# B&R Automation Studio project EFI (part 23)

#### SafetySample.var
```iecst
(********************************************************************
 * COPYRIGHT -- Bernecker + Rainer
 ********************************************************************
 * Program: SafetySample
 * File: SafetySample.var
 * Author: B&R
 ********************************************************************
 * Local variables of program SafetySample
 ********************************************************************)
VAR
	appcmd1 : DownloadCmdApplicationTypeV1; (*command structure for application download*)
	dataAcknMachineOptions : DownloadAcknMaOpTypeV1; (*data to acknowledge bit machine options*)
	datacmd1 : DownloadCmdMaOpTypeV1; (*command structure for machine options download*)
	datacmd2 : DownloadCmdExtMaOpTypeV1; (*command structure for extended machine options download*)
	dataMachineOptionsBitInput : ConfigurationBitOptionsTypeV1; (*data for bit machine options*)
	dataModuleFlagsInput : ConfigurationModuleFlagsTypeV1; (*data for module flags*)
	dialogApplication : BOOL; (*visualization dialog for application download*)
	dialogButtonLeft : BOOL; (*left button in visualization dialog*)
	dialogButtonRight : BOOL; (*right button in visualization dialog*)
	dialogData : BOOL; (*visualization dialog for machine options download*)
	dialogExtData : BOOL; (*visualization dialog for extended machine options download*)
	dialogRemoteCmd : BOOL; (*visualization dialog for remote control*)
	executeapp1 : BOOL; (*execute application download*)
	executedata1 : BOOL; (*execute machine options download*)
	executedata2 : BOOL; (*execute extended machine options download*)
	executeRemoteCmd : BOOL; (*execute remote control*)
	indexButtonLeft : UINT; (*index for button text*)
	indexButtonRight : UINT; (* index for button text*)
	indexCompareTextData : UINT; (*index for compare message machine options*)
	indexCompareTextExtData : UINT; (*index for compare message extended machine options*)
	indexFAILLed : UINT; (*index FAIL led*)
	indexFwAcknLed : UINT; (*index FW-ACKN led*)
	indexHeaderText : UINT; (*index dialog header text*)
	indexMessageText : UINT; (*index message text*)
	indexMxchgLed : UINT; (*index MXCHG led*)
	indexRELed : UINT; (*index R/E led*)
	Interface : STRING[80] := 'IF3'; (*interface information for SafeLOGIC*)
	Node : USINT := 10; (*node information for SafeLOGIC*)
	pDeviceListOut : REFERENCE TO ARRAY[0..1] OF ConfigurationDeviceTypeV1; (*device list from FUB*)
	pMachineOptionsBitOut : REFERENCE TO ConfigurationBitOptionsTypeV1; (*bit machine options from FUB*)
	pModuleFlagsOut : REFERENCE TO ConfigurationModuleFlagsTypeV1; (*module flags form FUB*)
	readUDIDhighSL : EplSDORead; (*function block to read UDID high from device*)
	readUDIDhighSLX : AsIOAccRead; (*function block to read UDID high from device*)
	readUDIDlowSL : EplSDORead; (*function block to read UDID low from device*)
	readUDIDlowSLX : AsIOAccRead; (*function block to read UDID low from device*)
	remotecmd : RemoteControlCmdTypeV1; (*command structure for remote control*)
	safeDownloadApplication_0 : safeDownloadApplication; (*function block safeDownloadApplication*)
	safeDownloadData_0 : safeDownloadData; (*function block safeDownloadData*)
	safeDownloadData_1 : safeDownloadData; (*function block safeDownloadData*)
	safeRemoteControl_0 : safeRemoteControl; (*function block safeRemoteControl*)
	slxused : BOOL; (*SafeLOGIC-X is used*)
	Station : STRING[80] := 'IF6.ST3'; (*station information for SafeLOGIC-X*)
	statusAcknInfoData : UINT; (*acknowledge boxes for machine options*)
	statusAcknInfoExtData : UINT; (*acknowledge boxes for extended machine options*)
	statusButtonActiv : ARRAY[0..15] OF USINT; (*button activ*)
	statusButtonInactiv : ARRAY[0..15] OF USINT; (*button inactiv*)
	statusButtonUnlockApp : UINT; (*unlock buttons application*)
	statusButtonUnlockData : UINT; (*unlock buttons data*)
	statusButtonUnlockExtData : UINT; (*unlock buttons extended data*)
	statusDialog : UINT; (*dialog box*)
	statusSetPassword : UINT; (*visualization status to set password*)
	statusSLInformation : UINT; (*display information for SafeLOGIC*)
	stautsSLXInformation : UINT; (*display information for SafeLOGIC-X*)
	UDID_High : UINT; (*UDID_high for SafelOGIC*)
	UDID_Low : UDINT; (*UDID_low for SafeLOGIC*)
	visuAcknExtData : DownloadAcknExtMaOpTypeV1; (*acknowledge extended machine options*)
	visuAcknMachineOptions : ARRAY[0..511] OF BOOL; (*acknowledge machine options*)
	visuApplicationCRC : STRING[8]; (*CRC HEX string for visualization*)
	visuDeviceListInput : ARRAY[0..1] OF DownloadDeviceTypeV1; (*device list input*)
	visuDeviceListOutput : ARRAY[0..1] OF DownloadDeviceTypeV1; (*device list output*)
	visuDintInput : ConfigurationDintOptionsTypeV1; (*DINT channels input*)
	visuDintOutput : ConfigurationDintOptionsTypeV1; (*DINT channels output*)
	visuEnableDINTOptions : BOOL; (*enable DINT options*)
	visuEnableINTOptions : BOOL; (*enable INT options*)
	visuEnableMachineOptions : BOOL; (*enable BIT options*)
	visuEnableModuleFlags : BOOL; (*enable module flags*)
	visuEnableUDINTOptions : BOOL; (*enable UDINT options*)
	visuEnableUINTOptions : BOOL; (*enable UINT options*)
	visuIntInput : ConfigurationIntOptionsTypeV1; (*INT channels input*)
	visuIntOutput : ConfigurationIntOptionsTypeV1; (*INT channels output*)
	visuMachineOptionsBitInput : ARRAY[0..511] OF BOOL; (*BIT options input*)
	visuMachineOptionsBitOutput : ARRAY[0..511] OF BOOL; (*BIT options output*)
	visuModuleFlagsNotPresentInput : ARRAY[0..1023] OF BOOL; (*not present module flags input*)
	visuModuleFlagsNotPresentOutput : ARRAY[0..1023] OF BOOL; (*not present module flags output*)
	visuModuleFlagsOptionalInput : ARRAY[0..1023] OF BOOL; (*optional module flags input*)
	visuModuleFlagsOptionalOutput : ARRAY[0..1023] OF BOOL; (*optional module flags output*)
	visuModuleFlagsStartupInput : ARRAY[0..1023] OF BOOL; (*startup module flags input*)
	visuModuleFlagsStartupOutput : ARRAY[0..1023] OF BOOL; (*startup module flags output*)
	visuUDID_High : STRING[8]; (*UDID hex string for visualization*)
	visuUDID_Low : STRING[8]; (*UDID hex string for visualization*)
	visuUdintInput : ConfigurationUdintOptionsTypeV1; (*UDINT channels input*)
	visuUdintOutput : ConfigurationUdintOptionsTypeV1; (*UDINT channels output*)
	visuUintInput : ConfigurationUintOptionsTypeV1; (*UINT channels input*)
	visuUintOutput : ConfigurationUintOptionsTypeV1; (*UINT channels output*)
	visuUsedSLIDData : UINT; (*SafeLOGIC ID for data download*)
	visuUsedSLIDRemote : UINT; (*SafeLOGIC ID for remote control*)
	xcnt : UINT; (*counter variable*)
	xEnableSafetyProgram : BOOL := FALSE; (*By default, it is not running*)
END_VAR
```

#### SafetySample.fun
```iecst
(********************************************************************
 * COPYRIGHT -- Bernecker + Rainer
 ********************************************************************
 * Program: SafetySample
 * File: SafetySample.fun
 * Author: B&R
 ********************************************************************
 * Functions and function blocks of program SafetySample
 ********************************************************************)

FUNCTION itoahex : UINT (*converts a UDINT values into a HEX character string*) (*$GROUP=User*)
	VAR_INPUT
		value : UDINT; (*UDINT value to be converted into a HEX character string*)
		pString : UDINT; (*pointer to the destination character string*)
	END_VAR
	VAR
		i_counter : USINT; (*internal variable*)
		i_value : UDINT; (*internal variable*)
		i_cvalue : USINT; (*internal variable*)
	END_VAR
END_FUNCTION
```

#### itoahex.st
```iecst
(********************************************************************
 * COPYRIGHT -- Bernecker + Rainer
 ********************************************************************
 * Program: SafetySample
 * File: itoahex.st
 * Author: B&R
 ********************************************************************
 * Implementation of program SafetySample
 ********************************************************************)

(* converts a UDINT values into a HEX character string *)
FUNCTION itoahex

	i_value := value;

	FOR i_counter := 0 TO 7 BY 1  DO
		i_cvalue := REAL_TO_USINT(brmfloor(UDINT_TO_REAL(i_value / REAL_TO_UDINT(EXPT(16, 7 - i_counter)))));
		IF i_cvalue = 0 THEN
			brsmemset(pString + i_counter, 48, 1); // 48 Dec = ASCII '0'
		ELSIF i_cvalue > 0 AND i_cvalue < 10 THEN
			brsitoa(i_cvalue, pString + i_counter);
		ELSIF i_cvalue >= 10 THEN
			brsmemset(pString + i_counter, i_cvalue + 55, 1); // 65 Dec = ASCII 'A'
		END_IF

		IF i_cvalue > 0 THEN
			i_value := i_value - REAL_TO_UDINT(EXPT(16, 7 - i_counter)) * i_cvalue;
		END_IF

	END_FOR

	itoahex := 0;

END_FUNCTION
```

#### SafetySample.st
```iecst
(********************************************************************
 * COPYRIGHT -- Bernecker + Rainer
 ********************************************************************
 * Program: SafetySample
 * File: SafetySample.st
 * Author: B&R
 ********************************************************************
 * Implementation of program SafetySample
 ********************************************************************)

PROGRAM _INIT

(* command structure for remote control FUB *)
remotecmd.Version := safeVERSION_R107;	(* version *)
remotecmd.Password := '';				(* password *)

(* command structure for application download *)
appcmd1.Version := safeVERSION_R107;	(* version *)
appcmd1.Password := '';					(* password *)
appcmd1.ApplicationID := 1;				(* application id *)

(* command structure for machine options download *)
datacmd1.Version := safeVERSION_R107;								(* version *)
datacmd1.Password := '';											(* password *)
datacmd1.pDeviceListInput := ADR(visuDeviceListInput);				(* device list *)
datacmd1.pMachineOptionsInput := ADR(dataMachineOptionsBitInput);	(* bit machine options *)
datacmd1.pModuleFlagsInput := ADR(dataModuleFlagsInput);			(* module flags *)
datacmd1.pAcknMachineOptions := ADR(dataAcknMachineOptions);		(* acknowledge information *)

(* command structure for extended machine options *)
datacmd2.Version := safeVERSION_R107;					(* version *)
datacmd2.Password := '';								(* password *)
datacmd2.pIntDataInput := ADR(visuIntInput);			(* INT channels *)
datacmd2.NumberIntInput := 1;							(* number of INT channels *)
datacmd2.pUintDataInput := ADR(visuUintInput);			(* UINT channels *)
datacmd2.NumberUintInput := 1;							(* number of UINT channels *)
datacmd2.pDintDataInput := ADR(visuDintInput);			(* DINT channels *)
datacmd2.NumberDintInput := 1;							(* number of DINT channels *)
datacmd2.pUdintDataInput := ADR(visuUdintInput);		(* UDINT channels *)
datacmd2.NumberUdintInput := 1;							(* number of UDINT channels *)
datacmd2.pAcknMachineOptions := ADR(visuAcknExtData);	(* acknowledge information *)

(* hide elements in visualization *)
FOR xcnt := 0 TO SIZEOF(statusButtonActiv) - 1 DO
	statusButtonActiv[xcnt] := 1;
END_FOR

(* hide elements in visualization *)
statusButtonUnlockApp := 1;
statusButtonUnlockData := 1;
statusAcknInfoData := 1;
statusButtonUnlockExtData := 1;
statusAcknInfoExtData := 1;
statusDialog := 1;

(* set SafeLOGIC ID *)
visuUsedSLIDRemote := 1;
visuUsedSLIDData := 1;

END_PROGRAM

PROGRAM _CYCLIC

	IF NOT xEnableSafetyProgram THEN
		RETURN;
	END_IF

	(****************************************************************************************************************************************)
	(****************************************************************************************************************************************)
	(****************************************************************************************************************************************)
	(* show dialog to ackn command *)
	IF (dialogRemoteCmd = 1) THEN
		statusDialog := 0;
		dialogRemoteCmd := 0;
		indexButtonLeft := 0;
		indexButtonRight := 1;
		indexHeaderText := 0;
		IF (remotecmd.Data = safeCMD_SK_FORMAT) THEN
			indexMessageText := 0;
		ELSIF (remotecmd.Data = safeCMD_SK_XCHG) THEN
			indexMessageText := 1;
		ELSIF (remotecmd.Data = safeCMD_1_UDID_ACKN) THEN
			indexMessageText := 2;
		ELSIF (remotecmd.Data = safeCMD_2_UDID_ACKN) THEN
			indexMessageText := 3;
		ELSIF (remotecmd.Data = safeCMD_3_UDID_ACKN) THEN
			indexMessageText := 4;
		ELSIF (remotecmd.Data = safeCMD_4_UDID_ACKN) THEN
			indexMessageText := 5;
		ELSIF (remotecmd.Data =  safeCMD_N_UDID_ACKN) THEN
			indexMessageText := 6;
		ELSIF (remotecmd.Data =  safeCMD_CLEAR_DATA) THEN
			indexMessageText := 7;
		ELSIF (remotecmd.Data = safeCMD_FW_ACKN) THEN
			indexMessageText := 8;
		ELSIF (remotecmd.Data = safeCMD_RESET) THEN
			indexMessageText := 9;
		END_IF
	END_IF

	(* if dialog is ackn execute fub *)
	IF (dialogButtonLeft = 1 AND indexHeaderText = 0) THEN
		executeRemoteCmd := 1;
		dialogButtonLeft := 0;
		statusDialog := 1;
	ELSIF (dialogButtonRight = 1 AND indexHeaderText = 0) THEN
		dialogButtonRight := 0;
		statusDialog := 1;
	END_IF

	(* password must be at least 6 characters long *)
	IF brsstrlen(ADR(remotecmd.NewPassword)) < 6 THEN
		statusSetPassword := 2;
	ELSE
		statusSetPassword := 0;
	END_IF

	safeRemoteControl_0(SafeLOGICID := visuUsedSLIDRemote, Execute := executeRemoteCmd, pCommandData := ADR(remotecmd));
	(* reset execution flag *)
	IF (safeRemoteControl_0.Done = 1 OR safeRemoteControl_0.Error = 1) THEN
		executeRemoteCmd := 0;
	END_IF

	(* variables for visualization *)
	IF (safeRemoteControl_0.SafeLOGICStatus.SafeKEYChanged = 1) THEN
		FOR xcnt := 0 TO SIZEOF(statusButtonActiv) - 1 DO
			statusButtonActiv[xcnt] := 1;
 			statusButtonInactiv[xcnt] := 0;
		END_FOR
		statusButtonActiv[1] := 0;
 		statusButtonInactiv[1] := 1;
	ELSIF (safeRemoteControl_0.SafeLOGICStatus.NumberOfUDIDMismatches = 1 AND safeRemoteControl_0.SafeLOGICStatus.Scanning = 0) THEN
		FOR xcnt := 0 TO SIZEOF(statusButtonActiv) - 1 DO
			statusButtonActiv[xcnt] := 1;
 			statusButtonInactiv[xcnt] := 0;
		END_FOR
		statusButtonActiv[3] := 0;
 		statusButtonInactiv[3] := 1;
	ELSIF (safeRemoteControl_0.SafeLOGICStatus.NumberOfUDIDMismatches = 2 AND safeRemoteControl_0.SafeLOGICStatus.Scanning = 0) THEN
		FOR xcnt := 0 TO SIZEOF(statusButtonActiv) - 1 DO
			statusButtonActiv[xcnt] := 1;
 			statusButtonInactiv[xcnt] := 0;
		END_FOR
		statusButtonActiv[4] := 0;
 		statusButtonInactiv[4] := 1;
	ELSIF (safeRemoteControl_0.SafeLOGICStatus.NumberOfUDIDMismatches = 3 AND safeRemoteControl_0.SafeLOGICStatus.Scanning = 0) THEN
		FOR xcnt := 0 TO SIZEOF(statusButtonActiv) - 1 DO
			statusButtonActiv[xcnt] := 1;
 			statusButtonInactiv[xcnt] := 0;
		END_FOR
		statusButtonActiv[5] := 0;
 		statusButtonInactiv[5] := 1;
	ELSIF (safeRemoteControl_0.SafeLOGICStatus.NumberOfUDIDMismatches = 4 AND safeRemoteControl_0.SafeLOGICStatus.Scanning = 0) THEN
		FOR xcnt := 0 TO SIZEOF(statusButtonActiv) - 1 DO
			statusButtonActiv[xcnt] := 1;
 			statusButtonInactiv[xcnt] := 0;
		END_FOR
		statusButtonActiv[6] := 0;
 		statusButtonInactiv[6] := 1;
	ELSIF (safeRemoteControl_0.SafeLOGICStatus.NumberOfUDIDMismatches > 4 AND safeRemoteControl_0.SafeLOGICStatus.Scanning = 0) THEN
		FOR xcnt := 0 TO SIZEOF(statusButtonActiv) - 1 DO
			statusButtonActiv[xcnt] := 1;
 			statusButtonInactiv[xcnt] := 0;
		END_FOR
		statusButtonActiv[7] := 0;
 		statusButtonInactiv[7] := 1;
	ELSIF (safeRemoteControl_0.SafeLOGICStatus.NumberOfDifferentFirmware <> 0 AND safeRemoteControl_0.SafeLOGICStatus.Scanning = 0) THEN
		FOR xcnt := 0 TO SIZEOF(statusButtonActiv) - 1 DO
			statusButtonActiv[xcnt] := 1;
 			statusButtonInactiv[xcnt] := 0;
		END_FOR
		statusButtonActiv[11] := 0;
 		statusButtonInactiv[11] := 1;
	ELSE
		FOR xcnt := 0 TO SIZEOF(statusButtonActiv) - 1 DO
			statusButtonActiv[xcnt] := 1;
 			statusButtonInactiv[xcnt] := 0;
		END_FOR
	END_IF
	(* status text - MXCHG *)
	IF (safeRemoteControl_0.SafeLOGICStatus.LedTestActive = 1) THEN
		indexMxchgLed := 40;
	ELSIF (safeRemoteControl_0.SafeLOGICStatus.Scanning = 1) THEN
		indexMxchgLed := 30;
	ELSIF (safeRemoteControl_0.SafeLOGICStatus.NumberOfUDIDMismatches = 1) THEN
		indexMxchgLed := 1;
	ELSIF (safeRemoteControl_0.SafeLOGICStatus.NumberOfUDIDMismatches = 2) THEN
		indexMxchgLed := 2;
	ELSIF (safeRemoteControl_0.SafeLOGICStatus.NumberOfUDIDMismatches = 3) THEN
		indexMxchgLed := 3;
	ELSIF (safeRemoteControl_0.SafeLOGICStatus.NumberOfUDIDMismatches = 4) THEN
		indexMxchgLed := 4;
	ELSIF (safeRemoteControl_0.SafeLOGICStatus.NumberOfUDIDMismatches > 4) THEN
		indexMxchgLed := 5;
	ELSIF (safeRemoteControl_0.SafeLOGICStatus.NumberOfMissingModules <> 0) THEN
		indexMxchgLed := 20;
	ELSIF (safeRemoteControl_0.SafeLOGICStatus.NumberOfUDIDMismatches = 0) THEN
		indexMxchgLed := 10;
	END_IF
	(* status text - FW-ACKN *)
	IF (safeRemoteControl_0.SafeLOGICStatus.SafeKEYChanged = 0 AND safeRemoteControl_0.SafeLOGICStatus.NumberOfDifferentFirmware = 0) THEN
		indexFwAcknLed := 10;
	ELSIF (safeRemoteControl_0.SafeLOGICStatus.SafeKEYChanged = 1) THEN
		indexFwAcknLed := 1;
	ELSIF (safeRemoteControl_0.SafeLOGICStatus.NumberOfDifferentFirmware <> 0) THEN
		indexFwAcknLed := 2;
	END_IF
	(* status text - FAIL *)
	IF (safeRemoteControl_0.SafeLOGICStatus.FailSafe <> 16#55) THEN
		indexFAILLed := 2;
	ELSIF (safeRemoteControl_0.SafeLOGICStatus.openSAFETYstate = 0) THEN
		indexFAILLed := 0;
	ELSIF (safeRemoteControl_0.SafeLOGICStatus.openSAFETYstate = 1) THEN
		indexFAILLed := 1;
	END_IF
	(* status text - R/E *)
	indexRELed := safeRemoteControl_0.SafeLOGICStatus.SafeOSState;

	(****************************************************************************************************************************************)
	(****************************************************************************************************************************************)
	(****************************************************************************************************************************************)
	(* show dialog to ackn command *)
	IF (dialogApplication = 1) THEN
		statusDialog := 0;
		dialogApplication := 0;
		indexButtonLeft := 0;
		indexButtonRight := 1;
		indexHeaderText := 1;
		indexMessageText := 10;
	END_IF

	(* if dialog is ackn unlock application *)
	IF (dialogButtonLeft = 1 AND indexHeaderText = 1) THEN
		appcmd1.Unlock := 1;
		dialogButtonLeft := 0;
		statusDialog := 1;
	ELSIF (dialogButtonRight = 1 AND indexHeaderText = 1) THEN
		appcmd1.Unlock := 2;
		dialogButtonRight := 0;
		statusDialog := 1;
	END_IF

	(* convert application CRC to HEX string *)
	itoahex(safeDownloadApplication_0.ApplicationCRC, ADR(visuApplicationCRC));

	safeDownloadApplication_0(SafeLOGICID := appcmd1.ApplicationID, Execute := executeapp1, pCommandData := ADR(appcmd1));

	(* show unlock button *)
	IF (safeDownloadApplication_0.UnlockRequired = 1) THEN
		statusButtonUnlockApp := 0;
	ELSE
		appcmd1.Unlock := 0;
		statusButtonUnlockApp := 1;
	END_IF

	(****************************************************************************************************************************************)
	(****************************************************************************************************************************************)
	(****************************************************************************************************************************************)
	(* disable machine options *)
	IF (visuEnableMachineOptions = FALSE) THEN
		datacmd1.pMachineOptionsInput := 0;
	ELSE
		datacmd1.pMachineOptionsInput := ADR(dataMachineOptionsBitInput);
	END_IF

	(* disable module flags *)
	IF (visuEnableModuleFlags = FALSE) THEN
		datacmd1.pModuleFlagsInput := 0;
	ELSE
		datacmd1.pModuleFlagsInput := ADR(dataModuleFlagsInput);
	END_IF

	(* Machine Option Bit #000 *)
	IF (visuMachineOptionsBitInput[0] = 1) THEN
		dataMachineOptionsBitInput.BitData[0].0 := 1;
	ELSE
		dataMachineOptionsBitInput.BitData[0].0 := 0;
	END_IF
	(* Machine Option Bit #001 *)
	IF (visuMachineOptionsBitInput[1] = 1) THEN
		dataMachineOptionsBitInput.BitData[0].1 := 1;
	ELSE
		dataMachineOptionsBitInput.BitData[0].1 := 0;
	END_IF
	(* Machine Option Bit #002 *)
	IF (visuMachineOptionsBitInput[2] = 1) THEN
		dataMachineOptionsBitInput.BitData[0].2 := 1;
	ELSE
		dataMachineOptionsBitInput.BitData[0].2 := 0;
	END_IF
	(* Optional Flag Module #1 *)
	IF (visuModuleFlagsOptionalInput[1] = 1) THEN
		dataModuleFlagsInput.Optional[0].1 := 1;
	ELSE
		dataModuleFlagsInput.Optional[0].1 := 0;
	END_IF
	(* Optional Flag Module #2 *)
	IF (visuModuleFlagsOptionalInput[2] = 1) THEN
		dataModuleFlagsInput.Optional[0].2 := 1;
	ELSE
		dataModuleFlagsInput.Optional[0].2 := 0;
	END_IF
	(* Startup Flag Module #1 *)
	IF (visuModuleFlagsStartupInput[1] = 1) THEN
		dataModuleFlagsInput.Startup[0].1 := 1;
	ELSE
		dataModuleFlagsInput.Startup[0].1 := 0;
	END_IF
	(* Startup Flag Module #2 *)
	IF (visuModuleFlagsStartupInput[2] = 1) THEN
		dataModuleFlagsInput.Startup[0].2 := 1;
	ELSE
		dataModuleFlagsInput.Startup[0].2 := 0;
	END_IF
	(* Not_Present Flag Module #1 *)
	IF (visuModuleFlagsNotPresentInput[1] = 1) THEN
		dataModuleFlagsInput.NotPresent[0].1 := 1;
	ELSE
		dataModuleFlagsInput.NotPresent[0].1 := 0;
	END_IF
	(* Not_Present Flag Module #2 *)
	IF (visuModuleFlagsNotPresentInput[2] = 1) THEN
		dataModuleFlagsInput.NotPresent[0].2 := 1;
	ELSE
		dataModuleFlagsInput.NotPresent[0].2 := 0;
	END_IF

	(* Ackn Machine Option Bit #000 *)
	IF (visuAcknMachineOptions[0] = 1) THEN
		dataAcknMachineOptions.AcknBitOptions[0].0 := 1;
	ELSE
		dataAcknMachineOptions.AcknBitOptions[0].0 := 0;
	END_IF
	(* Ackn Machine Option Bit #001 *)
	IF (visuAcknMachineOptions[1] = 1) THEN
		dataAcknMachineOptions.AcknBitOptions[0].1 := 1;
	ELSE
		dataAcknMachineOptions.AcknBitOptions[0].1 := 0;
	END_IF
	(* Ackn Machine Option Bit #002 *)
	IF (visuAcknMachineOptions[2] = 1) THEN
		dataAcknMachineOptions.AcknBitOptions[0].2 := 1;
	ELSE
		dataAcknMachineOptions.AcknBitOptions[0].2 := 0;
	END_IF

	(* show dialog to ackn command *)
	IF (dialogData = 1) THEN
		statusDialog := 0;
		dialogData := 0;
		indexButtonLeft := 0;
		indexButtonRight := 1;
		indexHeaderText := 2;
		indexMessageText := 11;
	END_IF

	(* if dialog is ackn unlock data *)
	IF (dialogButtonLeft = 1 AND indexHeaderText = 2) THEN
		datacmd1.Unlock := 1;
		dialogButtonLeft := 0;
		statusDialog := 1;
	ELSIF (dialogButtonRight = 1 AND indexHeaderText = 2) THEN
		datacmd1.Unlock := 2;
		dialogButtonRight := 0;
		statusDialog := 1;
	END_IF

	safeDownloadData_0(SafeLOGICID := visuUsedSLIDData, Execute := executedata1, Type:= safeDATA_TYPE_MAOP, pCommandData := ADR(datacmd1));

	(* data compare failed *)
	IF (safeDownloadData_0.StatusID = safeERR_DL_COMPARE_FAILED) THEN
		indexCompareTextData := 2;
	ELSE
		indexCompareTextData := 0;
	END_IF

	IF (safeDownloadData_0.UnlockRequired = 1) THEN
		(* data compare successful *)
		indexCompareTextData := 1;
		IF (datacmd1.pDeviceListOutput <> 0 AND datacmd1.NumberDevicesOutput <> 0) THEN
			pDeviceListOut ACCESS datacmd1.pDeviceListOutput;

			(* device #1 *)
			visuDeviceListOutput[0].SADR := pDeviceListOut[0].SADR;
			brsmemcpy(ADR(visuDeviceListOutput[0].UDID_High), ADR(pDeviceListOut[0].UDID[0]), 2);
			(* swap UDID *)
			visuDeviceListOutput[0].UDID_High := swapUINT(visuDeviceListOutput[0].UDID_High);
			brsmemcpy(ADR(visuDeviceListOutput[0].UDID_Low), ADR(pDeviceListOut[0].UDID[2]), 4);
			(* swap UDID *)
			visuDeviceListOutput[0].UDID_Low := swapUDINT(visuDeviceListOutput[0].UDID_Low);
			(* device #2 *)
			visuDeviceListOutput[1].SADR := pDeviceListOut[1].SADR;
			brsmemcpy(ADR(visuDeviceListOutput[1].UDID_High), ADR(pDeviceListOut[1].UDID[0]), 2);
			(* swap UDID *)
			visuDeviceListOutput[1].UDID_High := swapUINT(visuDeviceListOutput[1].UDID_High);
			brsmemcpy(ADR(visuDeviceListOutput[1].UDID_Low), ADR(pDeviceListOut[1].UDID[2]), 4);
			(* swap UDID *)
			visuDeviceListOutput[1].UDID_Low := swapUDINT(visuDeviceListOutput[1].UDID_Low);
		END_IF

		IF (datacmd1.pMachineOptionsOutput <> 0) THEN
			pMachineOptionsBitOut ACCESS datacmd1.pMachineOptionsOutput;

			(* Machine Option Bit #000 *)
			IF (pMachineOptionsBitOut.BitData[0].0 = 1) THEN
				visuMachineOptionsBitOutput[0] := 1;
			END_IF
			(* Machine Option Bit #001 *)
			IF (pMachineOptionsBitOut.BitData[0].1 = 1) THEN
				visuMachineOptionsBitOutput[1] := 1;
			END_IF
			(* Machine Option Bit #002 *)
			IF (pMachineOptionsBitOut.BitData[0].2 = 1) THEN
				visuMachineOptionsBitOutput[2] := 1;
			END_IF
		END_IF

		IF (datacmd1.pModuleFlagsOutput <> 0) THEN
			pModuleFlagsOut ACCESS datacmd1.pModuleFlagsOutput;

			(* Optional Flag Module #1 *)
			IF (pModuleFlagsOut.Optional[0].1 = 1) THEN
				visuModuleFlagsOptionalOutput[1] := 1;
			END_IF
			(* Optional Flag Module #2 *)
			IF (pModuleFlagsOut.Optional[0].2 = 1) THEN
				visuModuleFlagsOptionalOutput[2] := 1;
			END_IF
			(* Startup Flag Module #1 *)
			IF (pModuleFlagsOut.Startup[0].1 = 1) THEN
				visuModuleFlagsStartupOutput[1] := 1;
			END_IF
			(* Startup Flag Module #2 *)
			IF (pModuleFlagsOut.Startup[0].2 = 1) THEN
				visuModuleFlagsStartupOutput[2] := 1;
			END_IF
			(* Not_Present Flag Module #1 *)
			IF (pModuleFlagsOut.NotPresent[0].1 = 1) THEN
				visuModuleFlagsNotPresentOutput[1] := 1;
			END_IF
			(* Not_Present Flag Module #2 *)
			IF (pModuleFlagsOut.NotPresent[0].2 = 1) THEN
				visuModuleFlagsNotPresentOutput[2] := 1;
			END_IF
		END_IF
		(* show ackn box *)
		statusAcknInfoData := 0;
		(* show unlock button unlocked if one ACK is set *)
		IF (visuAcknMachineOptions[0] = 1 OR visuAcknMachineOptions[1] = 1 OR visuAcknMachineOptions[2] = 1) THEN
			statusButtonUnlockData := 0;
		END_IF
	ELSIF (safeDownloadData_0.Done = 1 OR safeDownloadData_0.Error = 1) THEN
		(* reset visualization elements *)
		brsmemset(ADR(visuDeviceListOutput), 0, SIZEOF(visuDeviceListOutput));
		brsmemset(ADR(visuMachineOptionsBitOutput), 0, SIZEOF(visuMachineOptionsBitOutput));
		brsmemset(ADR(visuModuleFlagsOptionalOutput), 0, SIZEOF(visuModuleFlagsOptionalOutput));
		brsmemset(ADR(visuModuleFlagsStartupOutput), 0, SIZEOF(visuModuleFlagsStartupOutput));
		brsmemset(ADR(visuModuleFlagsNotPresentOutput), 0, SIZEOF(visuModuleFlagsNotPresentOutput));
		(* hide ackn box *)
		statusAcknInfoData := 1;
		(* hide unlock button *)
		datacmd1.Unlock := 0;
		statusButtonUnlockData := 1;
		(* reset ackn flags *)
		visuAcknMachineOptions[0] := 0;
		visuAcknMachineOptions[1] := 0;
		visuAcknMachineOptions[2] := 0;
	ELSE
		(* hide ackn box *)
		statusAcknInfoData := 1;
		(* hide unlock button *)
		datacmd1.Unlock := 0;
		statusButtonUnlockData := 1;
	END_IF

	(****************************************************************************************************************************************)
	(****************************************************************************************************************************************)
	(****************************************************************************************************************************************)
	(* Enable for INT set *)
	IF (visuEnableINTOptions <> 0) THEN
		datacmd2.pIntDataInput := ADR(visuIntInput);
		datacmd2.NumberIntInput := 1;
	ELSE
		datacmd2.pIntDataInput := 0;
		datacmd2.NumberIntInput := 0;
	END_IF
	(* Enable for UINT set *)
	IF (visuEnableUINTOptions <> 0) THEN
		datacmd2.pUintDataInput := ADR(visuUintInput);
		datacmd2.NumberUintInput := 1;
	ELSE
		datacmd2.pUintDataInput := 0;
		datacmd2.NumberUintInput := 0;
	END_IF
	(* Enable for DINT set *)
	IF (visuEnableDINTOptions <> 0) THEN
		datacmd2.pDintDataInput := ADR(visuDintInput);
		datacmd2.NumberDintInput := 1;
	ELSE
		datacmd2.pDintDataInput := 0;
		datacmd2.NumberDintInput := 0;
	END_IF
	(* Enable for UDINT set *)
	IF (visuEnableUDINTOptions <> 0) THEN
		datacmd2.pUdintDataInput := ADR(visuUdintInput);
		datacmd2.NumberUdintInput := 1;
	ELSE
		datacmd2.pUdintDataInput := 0;
		datacmd2.NumberUdintInput := 0;
	END_IF

	(* show dialog to ackn command *)
	IF (dialogExtData = 1) THEN
		statusDialog := 0;
		dialogExtData := 0;
		indexButtonLeft := 0;
		indexButtonRight := 1;
		indexHeaderText := 3;
		indexMessageText := 11;
	END_IF

	(* if dialog is ackn unlock data *)
	IF (dialogButtonLeft = 1 AND indexHeaderText = 3) THEN
		datacmd2.Unlock := 1;
		dialogButtonLeft := 0;
		statusDialog := 1;
	ELSIF (dialogButtonRight = 1 AND indexHeaderText = 3) THEN
		datacmd2.Unlock := 2;
		dialogButtonRight := 0;
		statusDialog := 1;
	END_IF

	safeDownloadData_1(SafeLOGICID := visuUsedSLIDData, Execute := executedata2, Type:= safeDATA_TYPE_EXTMAOP, pCommandData := ADR(datacmd2));

	(* data compare failed *)
	IF (safeDownloadData_1.StatusID = safeERR_DL_COMPARE_FAILED) THEN
		indexCompareTextExtData := 2;
	ELSE
		indexCompareTextExtData := 0;
	END_IF

	IF (safeDownloadData_1.UnlockRequired = 1) THEN
		(* data compare successful *)
		indexCompareTextExtData := 1;

		(* INT channels *)
		IF (datacmd2.pIntDataOutput <> 0 AND datacmd2.NumberIntOutput <> 0) THEN
			brsmemcpy(ADR(visuIntOutput), datacmd2.pIntDataOutput, SIZEOF(visuIntOutput));
		END_IF
		(* UINT channels *)
		IF (datacmd2.pUintDataOutput <> 0 AND datacmd2.NumberUintOutput <> 0) THEN
			brsmemcpy(ADR(visuUintOutput), datacmd2.pUintDataOutput, SIZEOF(visuUintOutput));
		END_IF
		(* DINT channels *)
		IF (datacmd2.pDintDataOutput <> 0 AND datacmd2.NumberDintOutput <> 0) THEN
			brsmemcpy(ADR(visuDintOutput), datacmd2.pDintDataOutput, SIZEOF(visuDintOutput));
		END_IF
		(* UDINT channels *)
		IF (datacmd2.pUdintDataOutput <> 0 AND datacmd2.NumberUdintOutput <> 0) THEN
			brsmemcpy(ADR(visuUdintOutput), datacmd2.pUdintDataOutput, SIZEOF(visuUdintOutput));
		END_IF
		(* show ackn box *)
		statusAcknInfoExtData := 0;
		(* show unlock button if one ACK is set *)
		IF (visuAcknExtData.AcknIntOptions[0] = 1 OR visuAcknExtData.AcknUintOptions[0] = 1 OR visuAcknExtData.AcknDintOptions[0] = 1 OR visuAcknExtData.AcknUdintOptions[0] = 1) THEN
			statusButtonUnlockExtData := 0;
		END_IF
	ELSIF (safeDownloadData_1.Done = 1 OR safeDownloadData_1.Error = 1) THEN
		(* reset visualization elements *)
		brsmemset(ADR(visuIntOutput), 0, SIZEOF(visuIntOutput));
		brsmemset(ADR(visuUintOutput), 0, SIZEOF(visuUintOutput));
		brsmemset(ADR(visuDintOutput), 0, SIZEOF(visuDintOutput));
		brsmemset(ADR(visuUdintOutput), 0, SIZEOF(visuUdintOutput));
		(* hide ackn box *)
		statusAcknInfoExtData := 1;
		(* hide unlock button *)
		datacmd2.Unlock := 0;
		statusButtonUnlockExtData := 1;
		(* reset ackn flags *)
		visuAcknExtData.AcknIntOptions[0] := 0;
		visuAcknExtData.AcknUintOptions[0] := 0;
		visuAcknExtData.AcknDintOptions[0] := 0;
		visuAcknExtData.AcknUdintOptions[0] := 0;
	ELSE
		(* hide ackn box *)
		statusAcknInfoExtData := 1;
		(* hide unlock button *)
		datacmd2.Unlock := 0;
		statusButtonUnlockExtData := 1;
	END_IF

	(****************************************************************************************************************************************)
	(****************************************************************************************************************************************)
	(****************************************************************************************************************************************)
	(* read UDID from SafeLOGIC-X *)
	IF slxused = 1 THEN
		readUDIDlowSLX(enable := 1, pDeviceName := ADR(Station), pChannelName := ADR('UDID_low'));

		IF readUDIDlowSLX.status = 0 THEN
			UDID_Low := readUDIDlowSLX.value;
		ELSIF readUDIDlowSLX.status <> 65535 THEN
			UDID_Low := 0;
		END_IF

		readUDIDhighSLX(enable := 1, pDeviceName := ADR(Station), pChannelName := ADR('UDID_high'));

		IF readUDIDhighSLX.status = 0 THEN
			UDID_High := UDINT_TO_UINT(readUDIDhighSLX.value);
		ELSIF readUDIDhighSLX.status <> 65535 THEN
			UDID_High := 0;
		END_IF

		(* hide / show visualization elements *)
		stautsSLXInformation := 0;
		statusSLInformation := 1;
	(* read UDID form SafeLOGIC *)
	ELSE
		readUDIDlowSL(enable := 1, pDevice := ADR(Interface), node := Node, index := 16#2000, subindex := 6, pData := ADR(UDID_Low), datalen := SIZEOF(UDID_Low));

		IF readUDIDlowSL.status <> 0 AND readUDIDlowSL.status <> 65535 THEN
			UDID_Low := 0;
		END_IF

		readUDIDhighSL(enable := 1, pDevice := ADR(Interface), node := Node, index := 16#2000, subindex := 7, pData := ADR(UDID_High), datalen := SIZEOF(UDID_High));

		IF readUDIDhighSL.status <> 0 AND readUDIDhighSL.status <> 65535 THEN
			UDID_High := 0;
		END_IF

		(* hide / show visualization elements *)
		stautsSLXInformation := 1;
		statusSLInformation := 0;
	END_IF

	(* convert UDID to HEX string *)
	itoahex(UDID_Low, ADR(visuUDID_Low));
	itoahex(UDID_High, ADR(visuUDID_High));

	(****************************************************************************************************************************************)
	(****************************************************************************************************************************************)
	(****************************************************************************************************************************************)
	(* write UDID for SafeLOGIC to command structure *)
	appcmd1.UDID_Low := UDID_Low;
	appcmd1.UDID_High := UDID_High;
	datacmd1.UDID_Low := UDID_Low;
	datacmd1.UDID_High := UDID_High;
	datacmd2.UDID_Low := UDID_Low;
	datacmd2.UDID_High := UDID_High;

END_PROGRAM
```

- .gitignore (not shown)

### QA Notes.txt
```
This is the last folder for QA in the PLC project.
Below this folder, the QATestPLC repository have to be cloned to work properly
```

### Program Logical/UnitTest/Dryer/PrepareDryer (ANSIC) - Prepare the Machine to Start working

#### PrepareDryer.c - Groups test cases for addition
```c
/********************************************************************
 * COPYRIGHT -- Bernecker + Rainer
 ********************************************************************
 * Program: PrepareMachine
 * Author: Jorge Murria
 ********************************************************************
 * Prepare machine with basic test to allow proper behabior
 * and starting tasks
 ********************************************************************/

#include <bur/plctypes.h>

#ifdef _DEFAULT_INCLUDES
#include <AsDefault.h>
#endif

#include "UnitTest.h"

#include <stdio.h>
#include <unistd.h>
#include <time.h>         /* clock_t, clock, CLOCKS_PER_SEC */
#include <astime.h>

_LOCAL TIME TimeLast;
_LOCAL TIME endtime;
_LOCAL UDINT diff_t;
_LOCAL STRING stringAux[120];

#define FALSE 0
#define TRUE 1

void nextState(){
	exTimesPreFast = gDryer.St.exec.fast;
	exTimesPreSlow = gDryer.St.exec.slow;
	gTestsExec.iTestState++;
	TimeLast = clock_ms();
}

_TEST test_GoToZero(void)
{
	strcpy(gTestsExec.TestName, "test_GoToZero");
	switch (gTestsExec.iTestState)
	{
		case 0:
			gSimMachine.Commands.xToZero = TRUE;
			nextState();
			break;

		case 1:
			strcpy(gTestsExec.TestStateDesctiption, "Going to Zero");
			TEST_BUSY_CONDITION( !gDryer.St.Mode.xZero );
			nextState();
			break;

		case 2:
			gTestsExec.iTestState = 0;
			TEST_ASSERT(TRUE);
			TEST_DONE;
			break;

		default:
			break;
	}
}

_TEST test_PrepareBasicConfig(void)
{
	strcpy(gTestsExec.TestName, "test_PrepareBasicConfig");
	switch (gTestsExec.iTestState)
	{
		case 0:

			gDryer.Pt.SW.rBeltSpeedSetPoint = 15.0;	// 15.0m/min
			gDryer.Pt.SW.tiDelayConsent = SECONDS_TO_TIME(2);
			gDryer.In.xConsentOk = TRUE;

			gDryer.Pt.SW.Safety.rMaxBeltSpeedSetPoint = 70.0;
			gDryer.Pt.SW.Safety.rMarginSafePrint = 1.1;

			gBelt.parSw.rAxisLength = 650.0;
			gBelt.parSw.rGearBox = 35.0;

			gDryer.Pt.SW.xEnableNir = TRUE;

			gTransVacuum[1].Inputs.iPressureRaw = 16384; //This value is the equivalent to 0mbar of vacuum

			nextState();
			break;

		case 1:
			TEST_BUSY_CONDITION( gDryer.St.exec.fast < exTimesPreFast + 5 ); //We'll wait xx scan cycles
			nextState();
			break;

		case 2:
			gTestsExec.iTestState = 0;
			TEST_ASSERT(gDryer.Pt.xLeftHandMachine);
			TEST_DONE;
			break;

		default:
			break;
	}
}

_TEST test_GoToManualFromZero(void)
{
	strcpy(gTestsExec.TestName, "test_GoToManualFromZero");
	switch (gTestsExec.iTestState)
	{
		case 0:
			gSimMachine.Commands.xToZero = TRUE;
			nextState();
			break;

		case 1:
			strcpy(gTestsExec.TestStateDesctiption, "Going to Zero");
			TEST_BUSY_CONDITION( !gDryer.St.Mode.xZero );
			nextState();
			break;

		case 2:
			gSimMachine.Commands.xToManual = TRUE;
			nextState();
			break;

		case 3:
			strcpy(gTestsExec.TestStateDesctiption, "Going to Manual");
			TEST_BUSY_CONDITION( !gDryer.St.Mode.xManual );
			nextState();
			break;

		case 4:
			strcpy(gTestsExec.TestName, "test_PrepareMachine Finished!! Congrats!");
			strcpy(gTestsExec.TestStateDesctiption, "--");

			gTestsExec.iTestState = 0;
			TEST_ASSERT(TRUE);

			TEST_DONE;
			break;

		default:
			break;
	}
}

_TEST test_ReferenceManualMotors(void)
{
	if (gDryer.Pt.MachineModel != DryerType_NOZ2_NIR_ARCLAMP){
		iTestState = 0;
		TEST_DONE;
	}
	strcpy(gTestsExec.TestName, "test_ReferenceManualMotors");
	switch (gTestsExec.iTestState)
	{
		case 0:
			gSimMachine.Commands.xToManual = TRUE;
			nextState();
			break;

		case 1:
			strcpy(gTestsExec.TestStateDesctiption, "Going to Manual");
			TEST_BUSY_CONDITION( !gDryer.St.Mode.xManual );
			nextState();
			break;

		case 2:
			TEST_BUSY_CONDITION( gDryer.St.exec.fast < exTimesPreFast + 3 ); //We'll wait xx scan cycles
			gSimpleBlock[1].commands.xBarHomeOrder = TRUE;
			nextState();
			break;

		case 3:
			strcpy(gTestsExec.TestStateDesctiption, "Referencing vertical motors");
			TEST_BUSY_CONDITION( !gSimpleBlock[1].Status.Motor.xBarsHomed );
			nextState();
			break;

		case 4:
			gTestsExec.iTestState = 0;
			TEST_ASSERT(TRUE);

			strcpy(gTestsExec.TestName, "test_PrepareMachine Finished!! Congrats!");
			strcpy(gTestsExec.TestStateDesctiption, "--");

			TEST_DONE;
			break;

		default:
			break;
	}
}

/*
B+R UnitTest: This is generated code.
Do not edit! Do not move!
Description: UnitTest Testprogramm infrastructure (TestSet).
LastUpdated: 2021-05-20 08:42:32Z
By B+R UnitTest Helper Version: 2.0.1.59
*/
UNITTEST_FIXTURES(fixtures)
{
	new_TestFixture("test_GoToZero", test_GoToZero),
	new_TestFixture("test_PrepareBasicConfig", test_PrepareBasicConfig),
	new_TestFixture("test_GoToManualFromZero", test_GoToManualFromZero),
	new_TestFixture("test_ReferenceManualMotors", test_ReferenceManualMotors),
};

UNITTEST_CALLER_COMPLETE_EXPLICIT(PrepareDryer, "PrepareDryer", 0, 0, fixtures, 0, 0, 0);
```

#### PrepareDryer.var - PVs for the program and test suite
```iecst
(********************************************************************
 * COPYRIGHT -- Bernecker + Rainer
 ********************************************************************
 * Program: PrepareMachine
 * Author: Jorge Murria
 ********************************************************************
 * Local variables of program PrepareMachine
 * General variables - do not change
 ********************************************************************)
(*Describe the test*)
VAR
	Testsuite : UtMgrTestSuite := (Name:='PrepareDryer',Description:='Tests prepare the Dryer',Type:=utMgrTEST_TYPE_C,MetaInformation:='Some Meta Information can be added here');
END_VAR
(*Variables used in the tests*)
```

#### autoGeneratedFile.c - Auto generated code
```c
/*
B+R UnitTest: This is generated code.
Do not edit! Do not move!
Description: UnitTest Testprogramm infrastructure (List of TestSets).
LastUpdated: 2021-04-22 08:56:32Z
By B+R UnitTest Helper Version: 2.0.1.59
*/
#include "UnitTest.h"

UNITTEST_TESTSET_DECLARATION  PrepareDryer;

UNITTEST_TESTSET_FIXTURES(utTestSets)
{
	new_TestSet(PrepareDryer),
};
UNTITTEST_TESTSET_HANDLER();
```

### Program Logical/UnitTest/Dryer/BeltTests (ANSIC) - Belt related tests

#### autoGeneratedFile.c - Auto generated code
```c
/*
B+R UnitTest: This is generated code.
Do not edit! Do not move!
Description: UnitTest Testprogramm infrastructure (List of TestSets).
LastUpdated: 2019-11-08 11:44:31Z
By B+R UnitTest Helper Version: 2.0.1.59
*/
#include "UnitTest.h"

UNITTEST_TESTSET_DECLARATION  BeltTests;

UNITTEST_TESTSET_FIXTURES(utTestSets)
{
	new_TestSet(BeltTests),
};
UNTITTEST_TESTSET_HANDLER();
```

### Library Logical/UnitTest/Libraries/UnitTest (ANSIC, version 2.01.0) - Static library for UnitTest programs written in ANSI C /C++

#### Test.h
```c
/*
* Author: 		B+R
* Contents of this file are modified and extended
*/

/*
 * COPYRIGHT AND PERMISSION NOTICE
 *
 * Copyright (c) 2003 Embedded Unit Project
 *
 * All rights reserved.
 *
 * Permission is hereby granted, free of charge, to any person obtaining
 * a copy of this software and associated documentation files (the
 * "Software"), to deal in the Software without restriction, including
 * without limitation the rights to use, copy, modify, merge, publish,
 * distribute, and/or sell copies of the Software, and to permit persons
 * to whom the Software is furnished to do so, provided that the above
 * copyright notice(s) and this permission notice appear in all copies
 * of the Software and that both the above copyright notice(s) and this
 * permission notice appear in supporting documentation.
 *
 * THE SOFTWARE IS PROVIDED "AS IS", WITHOUT WARRANTY OF ANY KIND,
 * EXPRESS OR IMPLIED, INCLUDING BUT NOT LIMITED TO THE WARRANTIES OF
 * MERCHANTABILITY, FITNESS FOR A PARTICULAR PURPOSE AND NONINFRINGEMENT
 * OF THIRD PARTY RIGHTS. IN NO EVENT SHALL THE COPYRIGHT HOLDER OR
 * HOLDERS INCLUDED IN THIS NOTICE BE LIABLE FOR ANY CLAIM, OR ANY
 * SPECIAL INDIRECT OR CONSEQUENTIAL DAMAGES, OR ANY DAMAGES WHATSOEVER
 * RESULTING FROM LOSS OF USE, DATA OR PROFITS, WHETHER IN AN ACTION OF
 * CONTRACT, NEGLIGENCE OR OTHER TORTIOUS ACTION, ARISING OUT OF OR IN
 * CONNECTION WITH THE USE OR PERFORMANCE OF THIS SOFTWARE.
 *
 * Except as contained in this notice, the name of a copyright holder
 * shall not be used in advertising or otherwise to promote the sale,
 * use or other dealings in this Software without prior written
 * authorization of the copyright holder.
 *
 * $Id: Test.h,v 1.4 2004/02/10 16:19:29 arms22 Exp $
 */
#ifndef	__TEST_H__
#define	__TEST_H__

typedef struct __TestResult		TestResult;
typedef struct __TestResult	*TestResultRef;/*downward compatible*/

typedef struct __TestImplement	TestImplement;
typedef struct __TestImplement	*TestImplementRef;/*downward compatible*/

typedef enum testStatusEnum
{
    ut_BUSY = 0,
    ut_DONE = 1,
    ut_ABORT = 2
} testStatusEnum;

typedef char* 			(*TestNameFunction)(void *);

typedef testStatusEnum	(*TestRunFunction)(void *, TestResult *);
typedef int				(*TestCountTestCasesFunction)(void *);

typedef enum testStateEnum
{
    stateStart, 	/* print something */
    stateSetup,
    stateRun,
    stateTearDown,
    stateEnd,		/* print something */
    stateDefault, 	/* last state*/
} testStateEnum;

struct __TestImplement
{
	TestNameFunction 			name;
	TestRunFunction 			run;
	TestCountTestCasesFunction countTestCases;
};

typedef struct __Test	Test;
typedef struct __Test	*TestRef;/*downward compatible*/

struct __Test
{
	TestImplement *isa;
};

#define Test_name(s)			((Test*)s)->isa->name(s)
#define Test_run(s,r)			((Test*)s)->isa->run(s,r)
#define Test_countTestCases(s)	((Test*)s)->isa->countTestCases(s)

#endif/*__TEST_H__*/
```

#### TestCaller.h
```c
/*
* Author: 		B+R
* Contents of this file are modified and extended
*/

/*
 * COPYRIGHT AND PERMISSION NOTICE
 *
 * Copyright (c) 2003 Embedded Unit Project
 *
 * All rights reserved.
 *
 * Permission is hereby granted, free of charge, to any person obtaining
 * a copy of this software and associated documentation files (the
 * "Software"), to deal in the Software without restriction, including
 * without limitation the rights to use, copy, modify, merge, publish,
 * distribute, and/or sell copies of the Software, and to permit persons
 * to whom the Software is furnished to do so, provided that the above
 * copyright notice(s) and this permission notice appear in all copies
 * of the Software and that both the above copyright notice(s) and this
 * permission notice appear in supporting documentation.
 *
 * THE SOFTWARE IS PROVIDED "AS IS", WITHOUT WARRANTY OF ANY KIND,
 * EXPRESS OR IMPLIED, INCLUDING BUT NOT LIMITED TO THE WARRANTIES OF
 * MERCHANTABILITY, FITNESS FOR A PARTICULAR PURPOSE AND NONINFRINGEMENT
 * OF THIRD PARTY RIGHTS. IN NO EVENT SHALL THE COPYRIGHT HOLDER OR
 * HOLDERS INCLUDED IN THIS NOTICE BE LIABLE FOR ANY CLAIM, OR ANY
 * SPECIAL INDIRECT OR CONSEQUENTIAL DAMAGES, OR ANY DAMAGES WHATSOEVER
 * RESULTING FROM LOSS OF USE, DATA OR PROFITS, WHETHER IN AN ACTION OF
 * CONTRACT, NEGLIGENCE OR OTHER TORTIOUS ACTION, ARISING OUT OF OR IN
 * CONNECTION WITH THE USE OR PERFORMANCE OF THIS SOFTWARE.
 *
 * Except as contained in this notice, the name of a copyright holder
 * shall not be used in advertising or otherwise to promote the sale,
 * use or other dealings in this Software without prior written
 * authorization of the copyright holder.
 *
 * $Id: TestCaller.h,v 1.7 2004/02/10 16:19:29 arms22 Exp $
 */
#ifndef	__TESTCALLER_H__
#define	__TESTCALLER_H__

typedef struct __TestFixture	TestFixture;
typedef struct __TestFixture	*TestFixtureRef;/*downward compatible*/

struct __TestFixture
{
	const char *name;
	unsigned long mode;
	testStatusEnum (*test)(void);
};

#define new_TestFixture(name,test)\
	{\
		name,\
		1,\
		test\
	}

#define skipTestFixture(name,test)\
	{\
		name,\
		0,\
		test\
	}

typedef struct __TestCaller		TestCaller;
typedef struct __TestCaller	*TestCallerRef;/*downward compatible*/

struct __TestCaller
{
	TestImplement *isa;
	const  char					*name;
	testStateEnum 				state;
	char 						abort;
	testStatusEnum				(*setUp)(void);
	testStatusEnum				(*tearDown)(void);
	unsigned int 				numberOfFixtuers;
	TestFixture					*fixtuers;
	testStatusEnum				(*setUpSuite)(void);
	testStatusEnum				(*tearDownSuite)(void);
	/* per Set, called in each cycle */
	void 						(*cyclicSetCaller)(void);
	unsigned long				mode;
};

extern const TestImplement TestCallerImplement;

#define new_TestCaller(name,sup,tdw,numberOfFixtuers,fixtuers,setupSuite,teardownSuite, cyclicSuite )\
	{\
		(TestImplement*)&TestCallerImplement,\
		name,\
		stateStart,\
		0,\
		sup,\
		tdw,\
		numberOfFixtuers,\
		fixtuers,\
		setupSuite,\
		teardownSuite,\
		cyclicSuite,\
		1\
	}

#define skipTestCaller(name,sup,tdw,numberOfFixtuers,fixtuers,setupSuite,teardownSuite, cyclicSuite )\
	{\
		(TestImplement*)&TestCallerImplement,\
		name,\
		stateStart,\
		0,\
		sup,\
		tdw,\
		numberOfFixtuers,\
		fixtuers,\
		setupSuite,\
		teardownSuite,\
		cyclicSuite,\
		0\
	}

#endif/*__TESTCALLER_H__*/
```

#### TestListener.h
```c
/*
* Author: 		B+R
* Contents of this file are modified and extended
*/

/*
 * COPYRIGHT AND PERMISSION NOTICE
 *
 * Copyright (c) 2003 Embedded Unit Project
 *
 * All rights reserved.
 *
 * Permission is hereby granted, free of charge, to any person obtaining
 * a copy of this software and associated documentation files (the
 * "Software"), to deal in the Software without restriction, including
 * without limitation the rights to use, copy, modify, merge, publish,
 * distribute, and/or sell copies of the Software, and to permit persons
 * to whom the Software is furnished to do so, provided that the above
 * copyright notice(s) and this permission notice appear in all copies
 * of the Software and that both the above copyright notice(s) and this
 * permission notice appear in supporting documentation.
 *
 * THE SOFTWARE IS PROVIDED "AS IS", WITHOUT WARRANTY OF ANY KIND,
 * EXPRESS OR IMPLIED, INCLUDING BUT NOT LIMITED TO THE WARRANTIES OF
 * MERCHANTABILITY, FITNESS FOR A PARTICULAR PURPOSE AND NONINFRINGEMENT
 * OF THIRD PARTY RIGHTS. IN NO EVENT SHALL THE COPYRIGHT HOLDER OR
 * HOLDERS INCLUDED IN THIS NOTICE BE LIABLE FOR ANY CLAIM, OR ANY
 * SPECIAL INDIRECT OR CONSEQUENTIAL DAMAGES, OR ANY DAMAGES WHATSOEVER
 * RESULTING FROM LOSS OF USE, DATA OR PROFITS, WHETHER IN AN ACTION OF
 * CONTRACT, NEGLIGENCE OR OTHER TORTIOUS ACTION, ARISING OUT OF OR IN
 * CONNECTION WITH THE USE OR PERFORMANCE OF THIS SOFTWARE.
 *
 * Except as contained in this notice, the name of a copyright holder
 * shall not be used in advertising or otherwise to promote the sale,
 * use or other dealings in this Software without prior written
 * authorization of the copyright holder.
 *
 * $Id: TestListener.h,v 1.4 2004/02/10 16:19:29 arms22 Exp $
 */
#ifndef	__TESTLISTENER_H__
#define	__TESTLISTENER_H__

typedef struct __TestListnerImplement	TestListnerImplement;
typedef struct __TestListnerImplement	*TestListnerImplementRef;/*downward compatible*/

typedef void(*TestListnerStartTestCallBack)(void *,void *);
typedef void(*TestListnerEndTestCallBack)(void *,void *);
typedef void(*TestListnerSkippedTestCallBack)(void *,void *);

typedef void(*TestListnerAddFailureCallBack)(void *,void *,const char *,unsigned long,const char *);

typedef void(*TestListnerAddPassedCallBack)(void *,void *,const char *,unsigned long,const char *);
typedef void(*TestListnerAddInfoCallBack)(void *,void *,const char *,unsigned long,const char *);
typedef void(*TestListnerAddAbortCallBack)(void *,void *,const char *,unsigned long,const char *);
typedef void(*TestListnerLogCallBack)(void *,void *,const char *,unsigned long,const char *, signed short);

struct __TestListnerImplement
{
	TestListnerStartTestCallBack 	startTest;
	TestListnerEndTestCallBack 		endTest;
	TestListnerSkippedTestCallBack 	skippedTest;
	TestListnerAddFailureCallBack 	addFailure;
	TestListnerAddPassedCallBack 	addPassed;
	TestListnerAddInfoCallBack 		addInfo;
	TestListnerAddAbortCallBack 	addAbort;
	TestListnerLogCallBack			doLog;
};

/*typedef struct __TestListner	TestListner;*/	/*->TestResult.h*/
/*typedef struct __TestListner*	TestListnerRef;*/	/*->TestResult.h*/

struct __TestListner
{
	TestListnerImplement *isa;
};

#define TestListner_startTest(s,t)			((TestListner*)s)->isa->startTest(s,t)
#define TestListner_endTest(s,t)			((TestListner*)s)->isa->endTest(s,t)
#define TestListner_skippedTest(s,t)			((TestListner*)s)->isa->skippedTest(s,t)

#define TestListner_addFailure(s,t,m,l,f)	((TestListner*)s)->isa->addFailure(s,t,m,l,f)
#define TestListner_addPassed(s,t,m,l,f)	((TestListner*)s)->isa->addPassed(s,t,m,l,f)
#define TestListner_addInfo(s,t,m,l,f)		((TestListner*)s)->isa->addInfo(s,t,m,l,f)
#define TestListner_addAbort(s,t,m,l,f)		((TestListner*)s)->isa->addAbort(s,t,m,l,f)
#define TestListener_doLog(s,t,m,l,f,e)		if(s)(((TestListner*)s)->isa->doLog(s,t,m,l,f,e))
#endif/*__TESTLISTENER_H__*/
```

#### TestResult.h
```c
/*
* Author: 		B+R
* Contents of this file are modified and extended
*/

/*
* COPYRIGHT AND PERMISSION NOTICE
*
* Copyright (c) 2003 Embedded Unit Project
*
* All rights reserved.
*
* Permission is hereby granted, free of charge, to any person obtaining
* a copy of this software and associated documentation files (the
* "Software"), to deal in the Software without restriction, including
* without limitation the rights to use, copy, modify, merge, publish,
* distribute, and/or sell copies of the Software, and to permit persons
* to whom the Software is furnished to do so, provided that the above
* copyright notice(s) and this permission notice appear in all copies
* of the Software and that both the above copyright notice(s) and this
* permission notice appear in supporting documentation.
*
* THE SOFTWARE IS PROVIDED "AS IS", WITHOUT WARRANTY OF ANY KIND,
* EXPRESS OR IMPLIED, INCLUDING BUT NOT LIMITED TO THE WARRANTIES OF
* MERCHANTABILITY, FITNESS FOR A PARTICULAR PURPOSE AND NONINFRINGEMENT
* OF THIRD PARTY RIGHTS. IN NO EVENT SHALL THE COPYRIGHT HOLDER OR
* HOLDERS INCLUDED IN THIS NOTICE BE LIABLE FOR ANY CLAIM, OR ANY
* SPECIAL INDIRECT OR CONSEQUENTIAL DAMAGES, OR ANY DAMAGES WHATSOEVER
* RESULTING FROM LOSS OF USE, DATA OR PROFITS, WHETHER IN AN ACTION OF
* CONTRACT, NEGLIGENCE OR OTHER TORTIOUS ACTION, ARISING OUT OF OR IN
* CONNECTION WITH THE USE OR PERFORMANCE OF THIS SOFTWARE.
*
* Except as contained in this notice, the name of a copyright holder
* shall not be used in advertising or otherwise to promote the sale,
* use or other dealings in this Software without prior written
* authorization of the copyright holder.
*
* $Id: TestResult.h,v 1.7 2004/02/10 16:19:29 arms22 Exp $
*/
#ifndef	__TESTRESULT_H__
#define	__TESTRESULT_H__

#ifdef	__cplusplus
extern "C" {
#endif

/*typedef struct __TestResult		TestResult;*//* -> Test.h*/
/*typedef struct __TestResult*		TestResultRef;*//* -> Test.h*/

typedef struct __TestListner	TestListner;
typedef struct __TestListner	*TestListnerRef;/*downward compatible*/

struct __TestResult
{
	unsigned short runCount;
	unsigned short failureCount;
	unsigned short passedCount;
	unsigned short infoCount;
	unsigned short summarizedCount;
	unsigned short abortCount;
	unsigned short skippedTestCount;
	unsigned short suceessedTestCount;
	TestListner *listener;
};

#define new_TestResult(listener)\
{\
	0,\
	0,\
	0,\
	0,\
	0,\
	0,\
	0,\
	0,\
	(TestListner*)listener\
}

void TestResult_init(TestResult *self,TestListner *listner);
void TestResult_startTest(TestResult *self,Test *test);
void TestResult_endTest(TestResult *self,Test *test);
void TestResult_skipTest(TestResult *self,Test *test);

void TestResult_addFailure(TestResult *self,Test *test,const char *msg,unsigned long line,const char *file);
void TestResult_addPassed(TestResult *self,Test *test,const char *msg,unsigned long line,const char *file);
void TestResult_addInfo(TestResult *self,Test *test,const char *msg,unsigned long line,const char *file);
void TestResult_addAbort(TestResult *self,Test *test,const char *msg,unsigned long line,const char *file);

#ifdef	__cplusplus
}
#endif

#endif/*__TESTRESULT_H__*/
```

#### utRunner.h
```c
/********************************************************************
 * COPYRIGHT B+R
 ********************************************************************
 * Library: utRunner
 * File: utRunner.h
 * Author: B+R
 *******************************************************************/

#ifndef	__UT_RUNNER_H__
#define	__UT_RUNNER_H__

#include <bur/plctypes.h>

#include "UnitTest.h"
#include "UtMgr.h"
#include "include/TestCaller.h"

#ifdef __cplusplus
extern "C"
{
#endif

void utInit(UtMgrTestSuite_typ *TestSuiteRef);
void utCyclic(UtMgrTestSuite_typ *TestSuiteRef);
void utExit(UtMgrTestSuite_typ *TestSuiteRef);

#ifdef __cplusplus
};
#endif

#endif/*__UT_RUNNER_H__*/
```

### Library Logical/UnitTest/Libraries/LibAssert1 (ANSIC) - Sample library: Creation of custom asserts

#### LibAssert1_REAL_ArrayAsserts.c - Array of REAL: implementation of the assert
```c
/********************************************************************
 * COPYRIGHT -- Bernecker + Rainer
 ********************************************************************
 * Library: LibAssert1
 * File: LibAssert1_REAL_ArrayAsserts.c
 * Author: B+R
 *******************************************************************/

#include <bur/plctypes.h>

#include "asbrstr.h"
#include "LibAssert1_REAL_ArrayAsserts.h"

#define TRUE 1
#define FALSE 0

#define NR_OF_DETAILED_ENTRIES_TO_SHOW 10

/* Tests each REAL in the array for equality in range
Returns true if passed, false otherwise
delta: allowed tolerance (floats are not exact values)
expected: array of expected REAL values
acutal: array of REAL values under test
nrOfEntries: number of entries in array
line: location information
file: location information
*/
BOOL spl_assertImplRealArrayWithin(const REAL *delta,
                                   const REAL *expected, 	const REAL *actual, const unsigned long nrOfEntries,
                                   unsigned long line, const char *file)
{
	unsigned long i = 0;
	unsigned long countFail = 0;
	STRING buffer[100];
	STRING numbuf[30];

	/*------------------------------------------------------------*/
	for(i = 0; i < nrOfEntries; i++)
	{
		REAL diff = actual[i] - expected[i];
		REAL pos_delta = delta[i];

		if (diff < 0)
		{
			/* use absolute (positive) value */
			diff = 0.0f - diff;
		}
		if (pos_delta < 0)
		{
			/* use absolute (positive) value */
			pos_delta = 0.0f - pos_delta;
		}

		/* Check */
		if (pos_delta < diff)
		{
			/* count the failures */
			countFail++;

			/* for the first NR_OF_DETAILED_ENTRIES_TO_SHOW failures generate an informational message) */
			if(countFail < NR_OF_DETAILED_ENTRIES_TO_SHOW)
			{
				brsstrcpy((unsigned long) buffer, (unsigned long) "At array index ");
				brsitoa((int)i, (unsigned long)numbuf);
				brsstrcat((unsigned long) buffer, (unsigned long) numbuf);

				brsstrcat((unsigned long) buffer, (unsigned long) ": exp ");
				brsftoa((REAL)expected[i], (unsigned long)numbuf);
				brsstrcat((unsigned long) buffer, (unsigned long) numbuf);

				brsstrcat((unsigned long) buffer, (unsigned long)" was ");
				brsftoa((REAL)actual[i], (unsigned long)numbuf);
				brsstrcat((unsigned long) buffer, (unsigned long) numbuf);

				addInfo(buffer, line, file);
			}
		}
	}/* end for */
	/*------------------------------------------------------------*/
	/* All entries checked, generate notification for test report */
	if(0 == countFail)
	{
		addPassed("", line, file);
		return TRUE;
	}
	else
	{
		brsitoa(countFail, (unsigned long)numbuf);
		brsstrcpy((unsigned long)buffer, (unsigned long)numbuf);
		brsstrcat((unsigned long)buffer, (unsigned long)" failures occured in array ");
		addFailure(buffer, line, file);
		return FALSE;
	}
}

/* Tests each REAL in the array for equality
Returns true if passed, false otherwise
delta: allowed tolerance (floats are not exact values)
expected: array of expected REAL values
acutal: array of REAL values under test
nrOfEntries: number of entries in array
line: location information
file: location information
*/
BOOL spl_assertImplRealArrayEqual(const REAL delta,
                                  const REAL *expected, 	const REAL *actual, const unsigned long nrOfEntries,
                                  unsigned long line, const char *file)
{
	unsigned long i = 0;
	char countFail = 0;
	STRING buffer[100];
	STRING numbuf[30];

	/*------------------------------------------------------------*/
	for(i = 0; i < nrOfEntries; i++)
	{
		REAL diff = actual[i] - expected[i];
		REAL pos_delta = delta * (REAL)(expected[i]);

		if (diff < 0)
		{
			/* use absolute (positive) value */
			diff = 0.0f - diff;
		}
		if (pos_delta < 0)
		{
			/* use absolute (positive) value */
			pos_delta = 0.0f - pos_delta;
		}

		/* Check */
		if (pos_delta < diff)
		{
			/* count the failures */
			countFail++;

			/* for the first NR_OF_DETAILED_ENTRIES_TO_SHOW failures generate an informational message) */
			if(countFail < NR_OF_DETAILED_ENTRIES_TO_SHOW)
			{
				brsstrcpy((unsigned long) buffer, (unsigned long) "At array index ");
				brsitoa((int)i, (unsigned long) numbuf);
				brsstrcat((unsigned long) buffer, (unsigned long) numbuf);

				brsstrcat((unsigned long) buffer, (unsigned long) ": exp ");
				brsftoa((REAL)expected[i], (unsigned long)numbuf);
				brsstrcat((unsigned long) buffer, (unsigned long) numbuf);

				brsstrcat((unsigned long) buffer, (unsigned long) " was ");
				brsftoa((REAL)actual[i], (unsigned long)numbuf);
				brsstrcat((unsigned long) buffer, (unsigned long) numbuf);

				addInfo(buffer, 0, 0);
			}
		}
	}/* end for */

	/*------------------------------------------------------------*/
	/* All entries checked, generate notification for test report */
	if(0 == countFail)
	{
		addPassed("", line, file);
		return TRUE;
	}
	else
	{
		brsitoa(countFail, (unsigned long)numbuf);
		brsstrcpy((unsigned long)buffer, (unsigned long)numbuf);
		brsstrcat((unsigned long)buffer,(unsigned long) " failures occured in array ");
		addFailure(buffer, line, file);
		return FALSE;
	}
}
```

### Library Logical/UnitTest/Libraries/EFIAssert (ANSIC) - Sample library: Creation of custom asserts

#### EFIAssert.h
```c
/********************************************************************
 * COPYRIGHT -- Bernecker + Rainer
 ********************************************************************
 * Library: EFIAssert
 * File: EFIAssert.h
 * Author: EFI. Jorge Murria & Mihai Bront
 *
 *
 *  NOTE: If creating new custom assert librery, the folder has to be
 * included in the project in
 * Configuration/PLC(or PC_Any)/RightButton/Properties/Build/
 * and there in Adicional Include Directories
 *
 *******************************************************************/

#include <bur/plctypes.h>
#include "UnitTest.h"

/* When this file is included the defines, makros  of the following header files should be provided as well:  */

#include "EFIAssert_REAL_ArrayAsserts.h"
#include "EFIAssert_ThresholdAssert.h"
#include "EFIAssert_GreaterThanReal.h"
```

#### EFIAssert_REAL_ArrayAsserts.h
```c
/********************************************************************
 * COPYRIGHT -- Bernecker + Rainer
 ********************************************************************
 * Library: EFIAssert
 * File: EFIAssert_REAL_ArrayAsserts.h
 * Author: B+R
 *******************************************************************/

#include <bur/plctypes.h>
#include "UnitTest.h"

#ifdef __cplusplus
extern "C"
{
#endif

	/* Dummies for smart edit autocompletion.
	See below for the real macros used by the compiler  */
#ifdef _SMART_EDIT_DUMMY_

	/* This assert checks two arrays of floats for equality. TEST_FLOAT_PRECISION is used as default Delta.

	Note: An assert like this is generally more readable and meaningful than multiple TEST_ASSERT_EQUAL_FLOAT().
	It informs about how many entries failed in total and shows the first NR_OF_DETAILED_ENTRIES_TO_SHOW together with the array index the failure occured. */
	BOOL SPLEFI_ASSERT_ARRAY_EQUAL_REAL(REAL *expected[], REAL *actual[], UDINT nrOfEntries);

	/* This assert checks two arrays of floats for equality with an accepted delta per entry

	Note: An assert like this is generally more readable and meaningful than multiple TEST_ASSERT_FLOAT_WITHIN().
	It informs about how many entries failed in total and shows the first NR_OF_DETAILED_ENTRIES_TO_SHOW together with the array index the failure occured.
	*/
	BOOL SPLEFI_ASSERT_ARRAY_REAL_WITHIN(REAL *delta[], REAL *expected[], REAL *actual[], UDINT nrOfEntries);

#endif

	/*------------------------------------------------------------*/

	/* Prototyping of functions.
	These declaration of functions are used by the compiler to check number and type of arguments. */
	BOOL splefi_assertImplRealArrayEqual(const REAL delta,
	                                  const REAL *expected,
	                                  const REAL *actual,
	                                  const unsigned long nrOfEntries,
	                                  unsigned long line, const char *file);

	BOOL splefi_assertImplRealArrayWithin(const REAL *delta,
	                                   const REAL *expected,
	                                   const REAL *actual,
	                                   const unsigned long nrOfEntries,
	                                   unsigned long line, const char *file);

	/* Makros used in the test implementation.
	The macro passes the location information to the implemented assert. */

#define SPLEFI_ASSERT_ARRAY_EQUAL_REAL(expected, actual, nrOfEntries)	\
	splefi_assertImplRealArrayEqual((REAL)TEST_FLOAT_PRECISION, expected, actual, nrOfEntries, (unsigned long) __LINE__, __FILE__)

#define SPLEFI_ASSERT_ARRAY_REAL_WITHIN(delta, expected, actual, nrOfEntries)	\
	splefi_assertImplRealArrayWithin(delta, expected, actual, nrOfEntries,  (unsigned long) __LINE__, __FILE__)

#ifdef __cplusplus
};
#endif
```

#### EFIAssert_ThresholdAssert.c
```c
/********************************************************************
 * COPYRIGHT -- Bernecker + Rainer
 ********************************************************************
 * Library: EFIAssert
 * File: EFIAssert_ThresholdAssert.c
 * Author: B+R
 *******************************************************************/

#include <bur/plctypes.h>

#include "asbrstr.h"
#include "EFIAssert_ThresholdAssert.h"

#define TRUE 1
#define FALSE 0

/* Returns TRUE: Assert passed, FALSE otherwise
threshold: limit
actual: value under test
line: location information
file: location information
*/
BOOL splefi_assertUpperBoundary_DINT(const DINT threshold, const DINT actual,
                                  unsigned long line, const char *file)
{
	STRING buffer[100];
	STRING numbuf[15];

	/* Check */
	if(threshold > actual) /* Good case: actual value is below the allowed (expected) maximum. */
	{
		/* Inform the test framework about a passed assert*/
		addPassed("", line, file);
		return TRUE;
	}
	else /* Bad case: acutal value exceeded acceptable threshold  */
	{
		/* Generate message for failure */
		brsstrcpy((unsigned long) buffer, (unsigned long) "Limit ");
		brsitoa((int)threshold, (unsigned long)numbuf);
		brsstrcat((unsigned long) buffer, (unsigned long) numbuf);
		brsstrcat((unsigned long) buffer, (unsigned long) " exceeded (was ");

		brsitoa((int)actual, (unsigned long)numbuf);
		brsstrcat((unsigned long) buffer, (unsigned long) numbuf);
		brsstrcat((unsigned long) buffer, (unsigned long) " ) ");

		/* Add failure to test report */
		addFailure(buffer, line, file);
		return FALSE;
	}
};
```

### Program Logical/UnitTest/Tests/PrePrepare (ANSIC) - Prepare the Machine to Start working

#### autoGeneratedFile.c - Auto generated code
```c
/*
B+R UnitTest: This is generated code.
Do not edit! Do not move!
Description: UnitTest Testprogramm infrastructure (List of TestSets).
LastUpdated: 2023-06-16 09:04:29Z
By B+R UnitTest Helper Version: 2.0.1.59
*/
#include "UnitTest.h"

UNITTEST_TESTSET_DECLARATION  PrePrepare;

UNITTEST_TESTSET_FIXTURES(utTestSets)
{
	new_TestSet(PrePrepare),
};
UNTITTEST_TESTSET_HANDLER();
```

### Program Logical/UnitTest/Tests/PrepareMachine (ANSIC) - Prepare the Machine to Start working

#### PrepareMachine.c - Groups test cases for addition
```c
/********************************************************************
 * COPYRIGHT -- Bernecker + Rainer
 ********************************************************************
 * Program: PrepareMachine
 * Author: Jorge Murria
 ********************************************************************
 * Prepare machine with basic test to allow proper behabior
 * and starting tasks
 ********************************************************************/

#include <bur/plctypes.h>

#ifdef _DEFAULT_INCLUDES
#include <AsDefault.h>
#endif

#include "UnitTest.h"

#include <stdio.h>
#include <unistd.h>
#include <time.h>         /* clock_t, clock, CLOCKS_PER_SEC */
#include <astime.h>

_LOCAL TIME TimeLast;
_LOCAL TIME endtime;
_LOCAL UDINT diff_t;
_LOCAL STRING stringAux[120];

#define FALSE 0
#define TRUE 1

void nextState(){
	exTimesPreFast = gMachine.St.exec.fast;
	exTimesPreSlow = gMachine.St.exec.slow;
	iTestState++;
	TimeLast = clock_ms();
}

_TEST test_CheckMachine(void)
{
	strcpy(txTest, "test_CheckMachine");

	// Check txText <> than assigned, so just once
	if (strcmp(&txTest, &gSimMachine.Commands.LogTests.Text) != 0){
		strcpy(gSimMachine.Commands.LogTests.Text, txTest); gSimMachine.Commands.LogTests.xCommand = TRUE;
	}

	iTestState = 0;

	switch (gMachine.Pt.MachineModel)
	{
		case Type_P4_12B_L:
			TEST_ASSERT_EQUAL_INT(150, gMachine.St.iMachineModelCodeSW);
			TEST_DONE;
			break;

		case Type_P4_6B_L:
			TEST_ASSERT_EQUAL_INT(510, gMachine.St.iMachineModelCodeSW);
			TEST_DONE;
			break;

		case Type_SHLD:
			TEST_ASSERT_EQUAL_INT(3, gMachine.St.iMachineModelCodeSW);
			TEST_DONE;
			break;

		case Type_S1400:
			TEST_ASSERT_EQUAL_INT(14, gMachine.St.iMachineModelCodeSW);
			TEST_DONE;
			break;

		case Type_S1400_VAC_PWRLNK:
			TEST_ASSERT_EQUAL_INT(14, gMachine.St.iMachineModelCodeSW);
			TEST_DONE;
			break;

		case Type_S1400_VAC_CAN:
			TEST_ASSERT_EQUAL_INT(15, gMachine.St.iMachineModelCodeSW);
			TEST_DONE;
			break;

		case Type_NOZ_2_AQ:
			TEST_ASSERT_EQUAL_INT(39, gMachine.St.iMachineModelCodeSW);
			TEST_DONE;
			break;

		case Type_P5_OIL:
			TEST_ASSERT_EQUAL_INT(14, gMachine.St.iMachineModelCodeSW);
			TEST_DONE;
			break;

		case Type_P5_WTR:
			TEST_ASSERT_EQUAL_INT(14, gMachine.St.iMachineModelCodeSW);
			TEST_DONE;
			break;

		case Type_P4_CBK:
			TEST_ASSERT_EQUAL_INT(510, gMachine.St.iMachineModelCodeSW);
			TEST_DONE;
			break;

		case Type_NOZ_2_UV:
			TEST_ASSERT_EQUAL_INT(40, gMachine.St.iMachineModelCodeSW);
			TEST_DONE;
			break;

		case Type_NOZ_2_UV_White:
			TEST_ASSERT_EQUAL_INT(40, gMachine.St.iMachineModelCodeSW);
			TEST_DONE;
			break;

		case Type_CUBE:
			TEST_ASSERT_EQUAL_INT(1101, gMachine.St.iMachineModelCodeSW);
			TEST_DONE;
			break;

		case Type_CUBE_GULLIVER:
			TEST_ASSERT_EQUAL_INT(1102, gMachine.St.iMachineModelCodeSW);
			TEST_DONE;
			break;

		case Type_MECANO_UV_WHITE:
			TEST_ASSERT_EQUAL_INT(60, gMachine.St.iMachineModelCodeSW);
			TEST_DONE;
			break;

		case Type_MECANO_UV_OPV:
			TEST_ASSERT_EQUAL_INT(60, gMachine.St.iMachineModelCodeSW);
			TEST_DONE;
			break;

		case Type_MECANO_UV_WHITE_OPV:
			TEST_ASSERT_EQUAL_INT(60, gMachine.St.iMachineModelCodeSW);
			TEST_DONE;
			break;

		default:
			break;
	}
}

_TEST test_GoToZero(void)
{
	TEST_BUSY_CONDITION( gMachine.St.exec.fast < exTimesPreFast + 10 ); //We'll wait xx scan cycles
	strcpy(txTest, "test_GoToZero");
	if (strcmp(&txTest, &gSimMachine.Commands.LogTests.Text) != 0){
		strcpy(gSimMachine.Commands.LogTests.Text, txTest); gSimMachine.Commands.LogTests.xCommand = TRUE;
	}
	switch (iTestState)
	{
		case 0:
			gSimMachine.Commands.xToZero = TRUE;
			nextState();
			break;

		case 1:
			strcpy(txStateDesc, "Going to Zero");
			TEST_BUSY_CONDITION( !gMachine.St.Mode.xZero );
			nextState();
			break;

		case 2:
			iTestState = 0;
			TEST_ASSERT(TRUE);
			TEST_DONE;
			break;

		default:
			break;
	}
}

_TEST test_MachineLeft(void)
{
	TEST_BUSY_CONDITION( gMachine.St.exec.fast < exTimesPreFast + 10 ); //We'll wait xx scan cycles
	strcpy(txTest, "test_MachineLeft");
	if (strcmp(&txTest, &gSimMachine.Commands.LogTests.Text) != 0){
		strcpy(gSimMachine.Commands.LogTests.Text, txTest); gSimMachine.Commands.LogTests.xCommand = TRUE;
	}
	switch (iTestState)
	{
		case 0:
			gMachine.parSw.xMachineDirection = TRUE;
			nextState();
			break;

		case 1:
			TEST_BUSY_CONDITION( gMachine.St.exec.fast < exTimesPreFast + 5 ); //We'll wait xx scan cycles

			endtime = clock_ms();
			diff_t = difftime(endtime, TimeLast);
			UINT int_len;
			int_len = itoa(diff_t, &stringAux);
			strcpy(txTest, "this is the time ");
			strcat(&txTest, &stringAux);

			nextState();
			break;

		case 2:
			endtime = clock_ms();
			strcpy(txTest, "Waiting timer ");
			TEST_BUSY_CONDITION( endtime < TimeLast + 1 ); //We'll wait xx ms

			iTestState = 0;
			TEST_ASSERT_EQUAL_INT(gMachine.Pt.xLeftHandMachine, gMachine.parSw.xMachineDirection);
			TEST_DONE;
			break;

		default:
			break;
	}
}

_TEST test_PrepareBasicConfigLeft(void)
{
	TEST_BUSY_CONDITION( gMachine.St.exec.fast < exTimesPreFast + 10 ); //We'll wait xx scan cycles
	strcpy(txTest, "test_PrepareBasicConfig");
	if (strcmp(&txTest, &gSimMachine.Commands.LogTests.Text) != 0){
		strcpy(gSimMachine.Commands.LogTests.Text, txTest); gSimMachine.Commands.LogTests.xCommand = TRUE;
	}
	switch (iTestState)
	{
		case 0:
			gBlock[1].parSw.xEnableToMovements = TRUE;
			gBlock[1].parSw.xEnableToPrint = TRUE;
			gBlock[1].In.xWaterLevelSensor = TRUE;
			gBlock[1].In.xBarsIn = TRUE;

			gBlock[2].parSw.xEnableToMovements = (gMachine.Pt.CT.iNumBlocks>=2);
			gBlock[2].parSw.xEnableToPrint = (gMachine.Pt.CT.iNumBlocks>=2);
			gBlock[2].In.xWaterLevelSensor = (gMachine.Pt.CT.iNumBlocks>=2);
			gBlock[2].In.xBarsIn = TRUE;

			gMachine.parSw.Electronics.xRobotReadyL1 = TRUE;

			gMachine.parSw.rBeltSpeedSetPoint = 15.0;	// 15.0m/min
			gMachine.parSw.tiDelayConsent = SECONDS_TO_TIME(2);
			gMachine.In.xConsentL1Ok = TRUE;
			gMachine.In.xPowerSwitch = TRUE;

			gMachine.parSw.Safety.rMarginSafePrint = 1.1;
			gMachine.parSw.Safety.rMountedPieceOverthickness = 4.0;

			gMachine.parSw.Dtp.xDoubleLine = FALSE;

			gMachine.parSw.Clean.tiCleaningByTime = MINUTES_TO_TIME(12*60);
			gMachine.parSw.Clean.tiToCleanWhenPrinterStopped = MINUTES_TO_TIME(12*60);
			gMachine.parSw.Clean.iCleanMotorSpeedFwd = 5000;
			gMachine.parSw.Clean.iCleanMotorSpeedBwd = 5000;
			gMachine.parSw.Clean.iCleaningType = 1;
			gMachine.In.xSafetyEnabled = TRUE;
			gMachine.parSw.xAutoStartEnabled = FALSE;

			// Adding data for document
			gMachine.parSw.Hw.iMaxMediaLength = 9999;
			gMachine.parSw.Media.rLength = 1600;
			gMachine.parSw.Media.rWidth = 1400;
			if (gMachine.Pt.MachineModel == Type_CUBE){
				gMachine.parSw.Media.rGap = 3000;
			}
			else{
				gMachine.parSw.Media.rGap = 600;
			}
			gMachine.parSw.Media.rOffsetRegisterL1 = -700;
			gMachine.parSw.Media.rThickness = 2.0;

			//For machine models that detection system is defined by SW
			if (!gPhotoCells.status.xInstalled && !gDing.State.xDingInstalled){
				gMachine.parSw.Hw.xInstallnSensor = TRUE;
			}

			gBelt.parSw.rAxisLength = 650.0;
			gBelt.parSw.rGearBox = 10.0;

			gDing.In.xModuleOK = TRUE;
			gDing.In.xDingChannelFault = FALSE;
			gSimMachine.Commands.Media.rMediaThickness = 2;

			if (gPhotoCells.parameters.MotorType == STP_STEPPER){
				gPhotoCells.parSw.rThicknessReference = 12;
			}
			else{
				gPhotoCells.parSw.rThicknessReference = -12;
			}

			gPhotoCells.parSw.rMechOffset = -0.2;
			gPhotoCells.status.xBackModuleOk = TRUE;
			gPhotoCells.status.xFrontModuleOk = TRUE;

			gIclaSim[1].Parameters.SpeedFactor = 1.0;
			gIclaSim[2].Parameters.SpeedFactor = 1.0;
			gIclaSim[3].Parameters.SpeedFactor = 1.0;
			gIclaSim[4].Parameters.SpeedFactor = 1.0;
			gIclaSim[5].Parameters.SpeedFactor = 1.0;
			gIclaSim[6].Parameters.SpeedFactor = 1.0;
			gIclaSim[7].Parameters.SpeedFactor = 1.0;

			gTransVacuum[1].Inputs.iPressureRaw = 16384; //This value is the equivalent to 0mbar of vacuum
			gMachine.parSw.xJamDetectEnable = TRUE;
			//gEdgeHoldDown.parSw.xEnable = TRUE;

			//Line Configuration just if the machine has line
			if (gMachine.Pt.xControlledByLine) {
				gLine.Inputs.UPSs[1].LoadOnBattery = FALSE;
				gFeeder.Inputs.xModelInput[0]=TRUE;
				gFeeder.ParSw.xEnabled=TRUE;
				gPrimer.Inputs.xModelInput[0]=TRUE;
				gPrimer.ParSw.xEnabled=TRUE;
				gPrimer.ParSw.xEnablePriming=TRUE;
				if (gMachine.St.HwData.xIsWater) {
					gSarm.Inputs.xModelInput[0]=FALSE;
					gSarm.Parameters.xInstalled=FALSE;
					gSarm.ParSw.xEnabled=FALSE;
					gDryerAnc.Inputs.xModelInput[0]=TRUE;
					gDryerAnc.ParSw.xEnabled=TRUE;
					gDryerAnc.Inputs.xInRemote=TRUE;
				}
				else {
					gSarm.Inputs.xModelInput[0]=TRUE;
					gSarm.Parameters.xInstalled=TRUE;
					gSarm.ParSw.xEnabled=TRUE;
					gDryerAnc.Inputs.xModelInput[0]=FALSE;
					gDryerAnc.ParSw.xEnabled=FALSE;
					gDryerAnc.Inputs.xInRemote=FALSE;
				}
				gOverVarnish.Inputs.xModelInput[0]=TRUE;
				gOverVarnish.ParSw.xEnabled=gMachine.St.HwData.xIsWater;
				gOverVarnish.ParSw.xEnablePriming=TRUE;
				gStacker.Inputs.xModelInput[0]=TRUE;
				gStacker.ParSw.xEnabled=TRUE;

				//Variables needed to work with line properly
				gLine.Inputs.xPrinterPowered = TRUE;
				gLine.Inputs.xOvervoltageProtectionOk = TRUE;

				gSimMachine.Commands.Media.xMediaIfFeederFeeding = TRUE;
			}

			//Set safety
			gSimSafetyController.Commands.xSafetyToDefault = TRUE;

			//Curing leds
			for (iIndexPrepareCuring = 1; iIndexPrepareCuring <= gMachine.Pt.Hw.iMaxCuringLedBars; iIndexPrepareCuring++)
			{
				gCuringLed[iIndexPrepareCuring].Signals.Inputs.xFrontDoorClosed = TRUE;
				for (iIndexPsuOk = 1; iIndexPsuOk < 11; iIndexPsuOk++)
				{
					gCuringLed[iIndexPrepareCuring].Signals.Inputs.xPsuDcOk[iIndexPsuOk] = TRUE;
					gCuringLed[iIndexPrepareCuring].Signals.Inputs.xPsuAcOk[iIndexPsuOk] = TRUE;
				}

			}

			nextState();
			break;

		case 1:
			TEST_BUSY_CONDITION( gMachine.St.exec.fast < exTimesPreFast + 5 ); //We'll wait xx scan cycles
			nextState();
			break;

		case 2:
			iTestState = 0;
			if (gMachine.parSw.xMachineDirection){
				TEST_ASSERT(gMachine.Pt.xLeftHandMachine);
			}
			TEST_DONE;
			break;

		default:
			break;
	}
}

_TEST test_GoToManualFromZero(void)
{
	TEST_BUSY_CONDITION( gMachine.St.exec.fast < exTimesPreFast + 10 ); //We'll wait xx scan cycles
	strcpy(txTest, "test_GoToManualFromZero");
	if (strcmp(&txTest, &gSimMachine.Commands.LogTests.Text) != 0){
		strcpy(gSimMachine.Commands.LogTests.Text, txTest); gSimMachine.Commands.LogTests.xCommand = TRUE;
	}
	switch (iTestState)
	{
		case 0:
			gSimMachine.Commands.xToZero = TRUE;
			nextState();
			break;

		case 1:
			strcpy(txStateDesc, "Going to Zero");
			TEST_BUSY_CONDITION( !gMachine.St.Mode.xZero );
			nextState();
			break;

		case 2:
			gSimMachine.Commands.xToManual = TRUE;
			nextState();
			break;

		case 3:
			strcpy(txStateDesc, "Going to Manual");
			TEST_BUSY_CONDITION( !gMachine.St.Mode.xManual );
			nextState();
			break;

		case 4:
			iTestState = 0;
			TEST_ASSERT(TRUE);
			TEST_DONE;
			break;

		default:
			break;
	}
}

_TEST test_StartInks01(void)
{
	TEST_BUSY_CONDITION( gMachine.St.exec.fast < exTimesPreFast + 10 ); //We'll wait xx scan cycles
	strcpy(txTest, "test_StartInks01");
	if (strcmp(&txTest, &gSimMachine.Commands.LogTests.Text) != 0){
		strcpy(gSimMachine.Commands.LogTests.Text, txTest); gSimMachine.Commands.LogTests.xCommand = TRUE;
	}
	switch (iTestState)
	{
		case 0:
			//Activate the OK signal in all inputs and prepare parameters
			for (iIndexBlock = 1; iIndexBlock <= gMachine.Pt.CT.iNumBlocks; iIndexBlock++)
			{
				if(gBlock[iIndexBlock].parSw.xEnableToMovements){
					for (iIndex = 1; iIndex <= gBlock[iIndexBlock].parameters.Inks.iMaxBlockPrintBars; iIndex++)
					{
						gInks[iIndex].parSw.xEnabledBarToPrint = TRUE;
						gInks[iIndex].parSw.xColorLoadedInJob = TRUE;

						gInks[iIndex].parSw.Config.iMappingBar = iIndex;
						gInks[iIndex].parSw.xActTestMode = TRUE;
						gInks[iIndex].parSw.NegPump.rLowerLimMeniscusCritical = 0;
						gInks[iIndex].parSw.NegPump.rUpperLimMeniscusCritical = 70.0;
						gInks[iIndex].parSw.PosPump.rSetPoint = 7.0;
						gInks[iIndex].parSw.NegPump.rSetPointMeniscus = 24;
						gInks[iIndex].parSw.Temp.rSetPointTemp = 30.0;
						gInks[iIndex].parSw.tiDripTime = MILLISECONDS_TO_TIME(300*iIndex);

						gInksInputs[iIndex].xPrintHeadsPsuOK = TRUE;

						//Acknowledging whether chiller installed is related to inks system. Used later to execute some tests
						if(gInks[iIndex].parameters.InksChiller.iIndex > 0){
							iInksChillerIndex = gInks[iIndex].parameters.InksChiller.iIndex;
						}
					}
				}
			}

			//In uv machine model cases. Consider curing led bars mapping
			for (iIndexPrepareCuring = 1; iIndexPrepareCuring <= gMachine.Pt.Hw.iMaxCuringLedBars; iIndexPrepareCuring++)
			{
				if (gCuringLed[iIndexPrepareCuring].Parameters.xInstalled){
				//Checking were curing led is mapped and removing the ink bar mapped with his mapping index in previous lines
					gInks[gCuringLed[iIndexPrepareCuring].Parameters.iMappingBar].parSw.Config.iMappingBar = 0;
					gInks[gCuringLed[iIndexPrepareCuring].Parameters.iMappingBar].parSw.xEnabledBarToPrint = FALSE;
				}
			}

			//In case camera is installed, check its mapping to remove ink bar associated to that mapping previously
			if(gCamera.Parameters.xInstalled){
				gInks[gCamera.Parameters.iMappingBar].parSw.Config.iMappingBar = 0;
				gInks[gCamera.Parameters.iMappingBar].parSw.xEnabledBarToPrint = FALSE;
			}

			// Start inks
			for (iIndexBlock = 1; iIndexBlock <= gMachine.Pt.CT.iNumBlocks; iIndexBlock++)
			{
				if(gBlock[iIndexBlock].parSw.xEnableToMovements)
				{
					for (iIndex = 1; iIndex <= gBlock[iIndexBlock].parameters.Inks.iMaxBlockPrintBars; iIndex++)
					{
						if (gInks[iIndex].parSw.xEnabledBarToPrint){
							gInks[iIndex].ordersSw.xStartInks = TRUE;
							gInks[iIndex].ordersSw.xPowPrintHead = TRUE;
							iCheckInkStartedIndex = iIndex;
						}
					}
				}
			}

			nextState();
			break;

		case 1:
			strcpy(txStateDesc, "Starting Inks");
			TEST_BUSY_CONDITION( (gMachine.St.exec.fast < exTimesPreFast + 50) && INKS_STARTED != gInks[iCheckInkStartedIndex].status.iInkStateSw); //We'll wait xx scan cycles
			nextState();
			break;

		case 2:
			strcpy(txStateDesc, "Waiting to stabilize");
			TEST_BUSY_CONDITION( gMachine.St.exec.fast < exTimesPreFast + 50 ); //We'll wait xx scan cycles
			gMachine.In.Buttons.xReset = TRUE;
			nextState();
			break;

		case 3:
			strcpy(txStateDesc, "Resetting alarms");
			TEST_BUSY_CONDITION( gMachine.St.exec.fast < exTimesPreFast + 10 ); //We'll wait xx scan cycles
			TEST_ASSERT_EQUAL_INT(INKS_STARTED, gInks[iCheckInkStartedIndex].status.iInkStateSw);
			gMachine.In.Buttons.xReset = TRUE;
			nextState();
			break;

		case 4:
			strcpy(txStateDesc, "Remove reset button input");
			TEST_BUSY_CONDITION( gMachine.AlSummary.CurrentReasonStop[0]!=0 ); //We'll wait xx scan cycles
			gMachine.In.Buttons.xReset = FALSE;
			iTestState = 0;
			TEST_DONE;
			break;

		default:
			break;
	}
}

_TEST test_CalibrateThicknessSensorWithoutMedia(void)
{
	TEST_BUSY_CONDITION( gMachine.St.exec.fast < exTimesPreFast + 10 ); //We'll wait xx scan cycles

	//If the Test makes non sense, not execute it
	if (gPhotoCells.status.xInstalled){
		TEST_DONE;
	}
	strcpy(txTest, "test_CalibrateThicknessSensorWithoutMedia");
	if (strcmp(&txTest, &gSimMachine.Commands.LogTests.Text) != 0){
		strcpy(gSimMachine.Commands.LogTests.Text, txTest); gSimMachine.Commands.LogTests.xCommand = TRUE;
	}
	switch (iTestState)
	{
		case 0:
			gSimMachine.Commands.xToZero = TRUE;
			gDing.Parameters.xDingInstalled = TRUE;
			nextState();
			break;

		case 1:
			strcpy(txStateDesc, "Going to Zero");
			TEST_BUSY_CONDITION( !gMachine.St.Mode.xZero );
			nextState();
			break;

		case 2:
			gDing.In.xDingLow = FALSE;
			gDing.In.rHighDingMm = gDing.parSw.rCalibrationValue;
			gDing.Commands.xCalibrateThickness = TRUE;
			nextState();
			break;

		case 3:
			strcpy(txStateDesc, "Calibrating Analog Sensor");
			TEST_BUSY_CONDITION( gDing.Commands.xCalibrateThickness );
			nextState();
			break;

		case 4:
			iTestState = 0;
			TEST_ASSERT(!gDing.State.xDingReferenced);
			gDing.In.rHighDingMm = 0;
			TEST_DONE;
			break;

		default:
			break;
	}
}

_TEST test_CalibrateThicknessSensor(void)
{
	//If the Test makes non sense, not execute it
	if (gPhotoCells.status.xInstalled){
		TEST_DONE;
	}

	TEST_BUSY_CONDITION( gMachine.St.exec.fast < exTimesPreFast + 10 ); //We'll wait xx scan cycles

	strcpy(txTest, "test_CalibrateThicknessSensor");
	if (strcmp(&txTest, &gSimMachine.Commands.LogTests.Text) != 0){
		strcpy(gSimMachine.Commands.LogTests.Text, txTest); gSimMachine.Commands.LogTests.xCommand = TRUE;
	}
	switch (iTestState)
	{
		case 0:
			gSimMachine.Commands.xToZero = TRUE;
			gDing.Parameters.xDingInstalled = TRUE;
			nextState();
			break;

		case 1:
			strcpy(txStateDesc, "Going to Zero");
			TEST_BUSY_CONDITION( !gMachine.St.Mode.xZero );
			nextState();
			break;

		case 2:
			gDing.In.rHighDingMm = gDing.parSw.rCalibrationValue;
			gDing.In.xDingLow = TRUE;
			gDing.Commands.xCalibrateThickness = TRUE;
			nextState();
			break;

		case 3:
			strcpy(txStateDesc, "Calibrating Analog Sensor");
			TEST_BUSY_CONDITION( gDing.Commands.xCalibrateThickness );
			nextState();
			break;

		case 4:
			iTestState = 0;
			gDing.In.rHighDingMm = 0;
			gDing.In.xDingLow = FALSE;
			TEST_ASSERT(gDing.State.xDingReferenced);
			TEST_DONE;
			break;

		default:
			break;
	}
}

_TEST test_CalibrateNLaser(void)
{
	//If the Test makes non sense, not execute it
	if (!gPhotoCells.status.xInstalled || (gPhotoCells.status.xReferenced && iTestState==0)){
		TEST_DONE;
	}
	TEST_BUSY_CONDITION( gMachine.St.exec.fast < exTimesPreFast + 10 ); //We'll wait xx scan cycles

	strcpy(txTest, "test_CalibrateNLaser");
	if (strcmp(&txTest, &gSimMachine.Commands.LogTests.Text) != 0){
		strcpy(gSimMachine.Commands.LogTests.Text, txTest); gSimMachine.Commands.LogTests.xCommand = TRUE;
	}
	switch (iTestState)
	{
		case 0:
			gSimMachine.Commands.xToManual = TRUE;
			gMachine.In.Buttons.xReset = TRUE;
			nextState();
			break;

		case 1:
			strcpy(txStateDesc, "Going to Manual");
			TEST_BUSY_CONDITION( !gMachine.St.Mode.xManual );
			nextState();
			break;

		case 2:
			strcpy(txStateDesc, "Waiting to gear");
			TEST_BUSY_CONDITION(gPhotoCells.status.iSystemState != STP_GEARED && gPhotoCells.status.iSystemState != STP_STANDSTILL);
			gMachine.In.Buttons.xReset = FALSE;
			nextState();
			break;

		case 3:
			strcpy(txStateDesc, "Setting the sensors to false");
			//Remove all signals to allow reference
			for (iIndex = 0; iIndex < MAX_LAST_NSENSOR; iIndex++)
			{
				gPhotoCells.Inputs.Signals.xPhotoCells[iIndex] = FALSE;
			}
			gPhotoCells.commandsSw.xReference = TRUE;
			nextState();
			break;

		case 4:
			strcpy(txStateDesc, "Calibrating nLaserSensor");
			TEST_BUSY_CONDITION(gPhotoCells.commandsSw.xReference);
			nextState();
			break;

		case 5:
			strcpy(txStateDesc, "Going down searching Reference Sensor");
			TEST_BUSY_CONDITION( gMachine.St.exec.fast < exTimesPreFast + 5 ); //We'll wait xx scan cycles
			TEST_BUSY_CONDITION(gPhotoCells.status.xReferenced);
			TEST_BUSY_CONDITION(!gTransVacuum[1].Status.xAtSpeed && gTransVacuum[1].Status.xInstalled);
			TEST_BUSY_CONDITION( gMachine.St.exec.fast < exTimesPreFast + 5 );
			TEST_ASSERT(gPhotoCells.parameters.xHomingEnabled);
			nextState();
			break;

		case 6:
			strcpy(txStateDesc, "Waiting nsensor are referenced");
			TEST_BUSY_CONDITION( !gPhotoCells.status.xReferencing );
			if (gPhotoCells.status.xReferencing && !gPhotoCells.status.xReferenced && gTransVacuum[1].Parameters.xInstalled){
				TEST_BUSY_CONDITION( gMachine.St.exec.fast < exTimesPreFast + 5 );
				TEST_ASSERT(gTransVacuum[1].OrdersSw.xRunManual);
				TEST_ASSERT(gTransVacuum[1].parSw.rManSetPoint == 100.0);
			}
			nextState();
			break;

		case 7:
			strcpy(txStateDesc, "Going up searching Reference Sensor");
			TEST_BUSY_CONDITION( !gPhotoCells.status.xReferenced );
			TEST_BUSY_CONDITION( gMachine.St.exec.fast < exTimesPreFast + 5 ); //We'll wait xx scan cycles
			if (gPhotoCells.status.xReferencing && gPhotoCells.status.xReferenced && gTransVacuum[1].Parameters.xInstalled){
				TEST_BUSY_CONDITION( gMachine.St.exec.fast < exTimesPreFast + 5 );
				TEST_ASSERT(!gTransVacuum[1].OrdersSw.xRunManual);
			}
			nextState();
			break;

		case 8:
			strcpy(txStateDesc, "Waiting to finish referencing");
			TEST_BUSY_CONDITION( gMachine.St.exec.fast < exTimesPreFast + 5 ); //We'll wait xx scan cycles
			TEST_BUSY_CONDITION(gPhotoCells.status.iSystemState != STP_STANDSTILL);
			nextState();
			break;

		case 9:
			TEST_BUSY_CONDITION( gMachine.St.exec.fast < exTimesPreFast + 20 ); //We'll wait xx scan cycles
			TEST_ASSERT(gPhotoCells.status.xReferenced);
			TEST_ASSERT(!gTransVacuum[1].OrdersSw.xRunManual);
			iTestState = 0;
			TEST_DONE;
			break;

		default:
			break;
	}
}

_TEST test_ReferenceManualMotors(void)
{
	TEST_BUSY_CONDITION( gMachine.St.exec.fast < exTimesPreFast + 10 ); //We'll wait xx scan cycles
	strcpy(txTest, "test_ReferenceManualMotors");
	if (strcmp(&txTest, &gSimMachine.Commands.LogTests.Text) != 0){
		strcpy(gSimMachine.Commands.LogTests.Text, txTest); gSimMachine.Commands.LogTests.xCommand = TRUE;
	}
	switch (iTestState)
	{
		case 0:
			gSimMachine.Commands.xToManual = TRUE;
			nextState();
			break;

		case 1:
			strcpy(txStateDesc, "Going to Manual");
			TEST_BUSY_CONDITION( !gMachine.St.Mode.xManual );
			nextState();
			break;

		case 2:
			strcpy(txStateDesc, "Executing icla home order");
			gBlock[1].commands.xIclaHomeOrder = TRUE;
			gBlock[2].commands.xIclaHomeOrder = TRUE;
			nextState();
			break;

		case 3:
			strcpy(txStateDesc, "Referencing Iclas");
			TEST_BUSY_CONDITION( !gBlock[1].Status.Icla.xHomed || (!gBlock[2].Status.Icla.xHomed && gBlock[2].parameters.Hw.xExistBlock) );
			nextState();
			break;

		case 4:
			strcpy(txStateDesc, "Executing tray out order");
			gBlock[1].commands.Manual.xManTrayOut = TRUE;
			gBlock[2].commands.Manual.xManTrayOut = TRUE;
			nextState();
			break;

		case 5:
			strcpy(txStateDesc, "Moving the tray Out to enable referencing");
			TEST_BUSY_CONDITION( !gBlock[1].In.xTrayOut || (!gBlock[2].In.xTrayOut && gBlock[2].parameters.Hw.xExistBlock) );
			nextState();
			break;

		case 6:
			strcpy(txStateDesc, "Executing bar home order");
			gBlock[1].commands.xBarHomeOrder = TRUE;
			gBlock[2].commands.xBarHomeOrder = TRUE;
			nextState();
			break;

		case 7:
			strcpy(txStateDesc, "Referencing vertical motors");
			TEST_BUSY_CONDITION( !gBlock[1].Status.Motor.xBarsHomed || (!gBlock[2].Status.Motor.xBarsHomed && gBlock[2].parameters.Hw.xExistBlock) );
			nextState();
			break;

		case 8:
			iTestState = 0;
			TEST_ASSERT(TRUE);

			strcpy(txTest, "test_PrepareMachine Finished!! Congrats!");
			strcpy(txStateDesc, "--");

			TEST_DONE;
			break;

		default:
			break;
	}
}

_TEST test_ReferenceEhd(void)
{
	if (!gEdgeHoldDown.parameters.xInstalled || TRUE){
		TEST_DONE;
	}

	strcpy(txTest, "test_ReferenceEhd");
	switch (iTestState)
	{
		case 0:
			gSimMachine.Commands.xToZero = TRUE;
			nextState();
			break;

		case 1:
			strcpy(txStateDesc, "Going to Zero");
			TEST_BUSY_CONDITION( !gMachine.St.Mode.xZero );
			nextState();
			break;

		case 2:
			gSimMachine.Commands.xToAuto = TRUE;
			nextState();
			break;

		case 3:
			strcpy(txStateDesc, "Going to auto");
			TEST_BUSY_CONDITION( !gMachine.St.Mode.xAuto );
			nextState();
			break;

		case 4:
			TEST_BUSY_CONDITION( !gMachine.St.Position.xInCap );
			nextState();
			break;

		case 5:
			gSimMachine.Commands.xToZero = TRUE;
			nextState();
			break;

		case 6:
			strcpy(txStateDesc, "Going to Zero");
			TEST_BUSY_CONDITION( !gMachine.St.Mode.xZero );
			nextState();
			break;

		case 7:
			gSimMachine.Commands.xToManual = TRUE;
			TEST_BUSY_CONDITION( !gMachine.St.Mode.xManual );
			nextState();
			break;

		case 8:
			TEST_BUSY_CONDITION( gEdgeHoldDown.status.iSystemState!= EHD_MANUAL );
			TEST_BUSY_CONDITION( gPairedMotors[1].status.iSystemState != STANDSTILL );
			TEST_BUSY_CONDITION( gPairedMotors[2].status.iSystemState != STANDSTILL );
			gEdgeHoldDown.commandsSw.xReference = TRUE;
			nextState();
			break;

		case 9:
			strcpy(txStateDesc, "Referencing EHD motors");
			TEST_BUSY_CONDITION( !gEdgeHoldDown.status.xReferenced );
			TEST_ASSERT(gEdgeHoldDown.status.xReferenced);
			TEST_ASSERT(gPairedMotors[1].Motor[1].rPositionMotor==gPairedMotors[1].Motor[2].rPositionMotor);
			TEST_ASSERT(gPairedMotors[1].Motor[1].rPositionMotor==gPairedMotors[1].parameters.rMechPositionMin);
			TEST_ASSERT(gPairedMotors[2].Motor[1].rPositionMotor==gPairedMotors[2].Motor[2].rPositionMotor);
			TEST_ASSERT(gPairedMotors[2].Motor[1].rPositionMotor==gPairedMotors[2].parameters.rMechPositionMin);
			strcpy(txStateDesc, "Disabling ehd");
			gEdgeHoldDown.parSw.xEnable=FALSE;
			gSimMachine.Commands.xToZero = TRUE;
			TEST_BUSY_CONDITION( !gMachine.St.Mode.xZero );

			nextState();
			break;

		case 10:
			strcpy(txStateDesc, "Setting ehd to resting position when disabled");
			gSimMachine.Commands.xToAuto = TRUE;
			TEST_BUSY_CONDITION( !gMachine.St.Mode.xAuto );
			TEST_BUSY_CONDITION(gEdgeHoldDown.status.xEnabled);
			TEST_ASSERT(!gEdgeHoldDown.status.xEnabled);

			nextState();
			break;

		case 11:
			iTestState = 0;

			strcpy(txTest, "test_PrepareMachine Finished!! Congrats!");
			strcpy(txStateDesc, "--");

			TEST_DONE;
			break;

		default:
			break;
	}
}

/*
B+R UnitTest: This is generated code.
Do not edit! Do not move!
Description: UnitTest Testprogramm infrastructure (TestSet).
LastUpdated: 2023-05-16 08:14:57Z
By B+R UnitTest Helper Version: 2.0.1.59
*/
UNITTEST_FIXTURES(fixtures)
{
	new_TestFixture("test_CheckMachine", test_CheckMachine),
	new_TestFixture("test_GoToZero", test_GoToZero),
	new_TestFixture("test_MachineLeft", test_MachineLeft),
	new_TestFixture("test_PrepareBasicConfigLeft", test_PrepareBasicConfigLeft),
	new_TestFixture("test_GoToManualFromZero", test_GoToManualFromZero),
	new_TestFixture("test_StartInks01", test_StartInks01),
	new_TestFixture("test_CalibrateThicknessSensorWithoutMedia", test_CalibrateThicknessSensorWithoutMedia),
	new_TestFixture("test_CalibrateThicknessSensor", test_CalibrateThicknessSensor),
	new_TestFixture("test_CalibrateNLaser", test_CalibrateNLaser),
	new_TestFixture("test_ReferenceManualMotors", test_ReferenceManualMotors),
	new_TestFixture("test_ReferenceEhd", test_ReferenceEhd),
};

UNITTEST_CALLER_COMPLETE_EXPLICIT(PrepareMachine, "PrepareMachine", 0, 0, fixtures, 0, 0, 0);
```

#### PrepareMachine.var - PVs for the program and test suite
```iecst
(********************************************************************
 * COPYRIGHT -- Bernecker + Rainer
 ********************************************************************
 * Program: PrepareMachine
 * Author: Jorge Murria
 ********************************************************************
 * Local variables of program PrepareMachine
 * General variables - do not change
 ********************************************************************)
(*Describe the test*)
VAR
	Testsuite : UtMgrTestSuite := (Name:='PrepareMachine',Description:='Tests prepare the Machine ',Type:=utMgrTEST_TYPE_C,MetaInformation:='Some Meta Information can be added here');
END_VAR
(*Variables used in the tests*)
```

#### testSuite.c - Handling of program and test suite
```c
/********************************************************************
 * COPYRIGHT -- Bernecker + Rainer
 ********************************************************************
 * Program: PrepareMachine
 * Author: B+R
 ********************************************************************
 * Test registration and handshake
 ********************************************************************/

#include <bur/plctypes.h>

#ifdef _DEFAULT_INCLUDES
#include <AsDefault.h>
#endif

#include "UnitTest.h"

void _INIT initTestSuite(void)
{
	utInit(&Testsuite);
}

void _CYCLIC cyclicWithTest(void)
{
	utCyclic(&Testsuite);
}

void _EXIT exitTestSuite(void)
{
	utExit(&Testsuite);
}
```

### Program Logical/UnitTest/Tests/BeltTests (ANSIC) - Belt related tests
